KUKA KRL program: firepit2_2.src

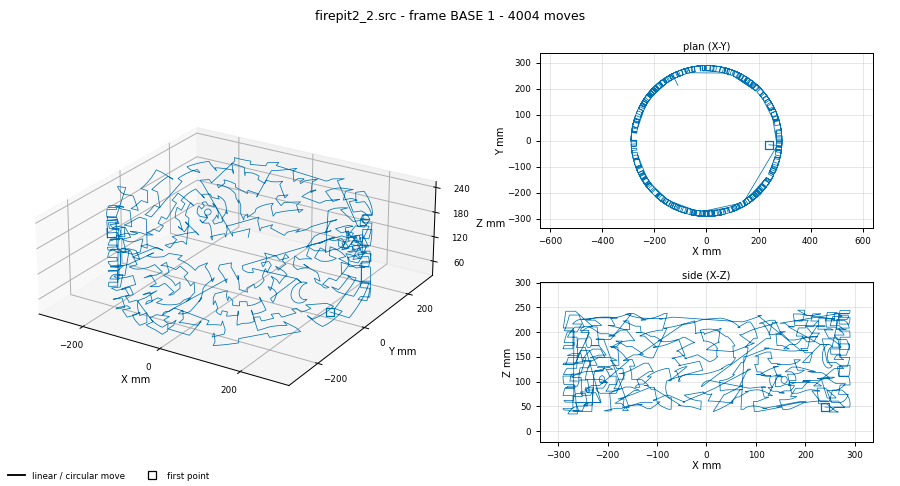
[picture p0: tool path of firepit2_2.src in frame BASE 1, 4004 of 4006 moves have a stored position in this frame; points joined in program order, loops and branches not executed]
&ACCESS RVP
&REL 1
&PARAM TEMPLATE = C:\KRC\Roboter\Template\vorgabe
&PARAM EDITMASK = *
DEF firepit2_2( )
EXT BAS (BAS_COMMAND :IN,REAL :IN )
DECL EKI_STATUS RET

INT INDX
FOR INDX=1 TO 6
	$ACC_AXIS[INDX]=50
	$VEL_AXIS[INDX]=20
ENDFOR

$VEL.ORI1=200
$VEL.ORI2=200
$ACC.ORI1=100
$ACC.ORI2=100

$VEL.CP = 0.1

$ACC.CP = 1

$IPO_MODE = #TCP
$APO.CDIS = 0.5
$ADVANCE = 5

$ACT_TOOL = 1
$TOOL=TOOL_DATA[1]
$ACT_BASE = 1
$BASE=BASE_DATA[1]

RET=EKI_Init("oxy")
RET=EKI_Open("oxy")

RET=EKI_SetBool("oxy","torchState",FALSE)
RET = EKI_Send("oxy","torchState")
PTP {A1 0.0,A2 -100.0,A3 150.0,A4 0.0,A5 -50.0,A6 0.0}

LIN {X 239.531,Y -14.995,Z 48.357,A 176.418,B 90.000,C 0.000} C_DIS
LIN {X 287.437,Y -17.994,Z 48.357,A 176.418,B 90.000,C 0.000} C_DIS
LIN {X 289.433,Y -18.119,Z 48.357,A 176.418,B 90.000,C 0.000} C_DIS
WAIT SEC 1.75
RET=EKI_SetBool("oxy","torchState",TRUE)
RET = EKI_Send("oxy","torchState")
LIN {X 289.566,Y -15.777,Z 49.221,A 176.881,B 90.000,C 0.000} C_DIS
LIN {X 289.684,Y -13.432,Z 50.078,A 177.345,B 90.000,C 0.000} C_DIS
LIN {X 289.787,Y -11.084,Z 50.930,A 177.810,B 90.000,C 0.000} C_DIS
LIN {X 289.865,Y -8.732,Z 51.772,A 178.274,B 90.000,C 0.000} C_DIS
LIN {X 289.925,Y -6.377,Z 52.608,A 178.740,B 90.000,C 0.000} C_DIS
LIN {X 289.970,Y -4.020,Z 53.438,A 179.206,B 90.000,C 0.000} C_DIS
LIN {X 289.992,Y -1.659,Z 54.260,A 179.672,B 90.000,C 0.000} C_DIS
LIN {X 289.994,Y 0.704,Z 55.074,A -179.861,B 90.000,C 0.000} C_DIS
LIN {X 289.981,Y 3.069,Z 55.883,A -179.394,B 90.000,C 0.000} C_DIS
LIN {X 289.946,Y 5.437,Z 56.685,A -178.926,B 90.000,C 0.000} C_DIS
LIN {X 289.890,Y 7.807,Z 57.478,A -178.457,B 90.000,C 0.000} C_DIS
LIN {X 289.818,Y 10.178,Z 58.266,A -177.989,B 90.000,C 0.000} C_DIS
LIN {X 289.726,Y 12.550,Z 59.048,A -177.520,B 90.000,C 0.000} C_DIS
LIN {X 289.610,Y 14.925,Z 59.821,A -177.050,B 90.000,C 0.000} C_DIS
LIN {X 289.480,Y 17.300,Z 60.589,A -176.580,B 90.000,C 0.000} C_DIS
LIN {X 289.329,Y 19.676,Z 61.350,A -176.110,B 90.000,C 0.000} C_DIS
LIN {X 289.155,Y 22.053,Z 62.103,A -175.639,B 90.000,C 0.000} C_DIS
LIN {X 288.966,Y 24.431,Z 62.851,A -175.167,B 90.000,C 0.000} C_DIS
LIN {X 288.755,Y 26.809,Z 63.592,A -174.696,B 90.000,C 0.000} C_DIS
LIN {X 288.522,Y 29.187,Z 64.326,A -174.224,B 90.000,C 0.000} C_DIS
LIN {X 288.274,Y 31.565,Z 65.055,A -173.751,B 90.000,C 0.000} C_DIS
LIN {X 288.003,Y 33.943,Z 65.776,A -173.278,B 90.000,C 0.000} C_DIS
LIN {X 287.711,Y 36.321,Z 66.491,A -172.805,B 90.000,C 0.000} C_DIS
LIN {X 287.405,Y 38.698,Z 67.201,A -172.331,B 90.000,C 0.000} C_DIS
LIN {X 287.072,Y 41.074,Z 67.903,A -171.857,B 90.000,C 0.000} C_DIS
LIN {X 286.721,Y 43.449,Z 68.599,A -171.383,B 90.000,C 0.000} C_DIS
LIN {X 286.357,Y 45.823,Z 69.290,A -170.909,B 90.000,C 0.000} C_DIS
LIN {X 285.961,Y 48.195,Z 69.973,A -170.433,B 90.000,C 0.000} C_DIS
LIN {X 285.553,Y 50.566,Z 70.651,A -169.958,B 90.000,C 0.000} C_DIS
LIN {X 285.125,Y 52.936,Z 71.323,A -169.482,B 90.000,C 0.000} C_DIS
LIN {X 284.672,Y 55.302,Z 71.988,A -169.006,B 90.000,C 0.000} C_DIS
LIN {X 284.205,Y 57.668,Z 72.649,A -168.530,B 90.000,C 0.000} C_DIS
LIN {X 283.714,Y 60.030,Z 73.302,A -168.053,B 90.000,C 0.000} C_DIS
LIN {X 283.203,Y 62.390,Z 73.949,A -167.576,B 90.000,C 0.000} C_DIS
LIN {X 282.679,Y 64.747,Z 74.593,A -167.099,B 90.000,C 0.000} C_DIS
LIN {X 282.124,Y 67.101,Z 75.228,A -166.621,B 90.000,C 0.000} C_DIS
LIN {X 281.556,Y 69.452,Z 75.859,A -166.143,B 90.000,C 0.000} C_DIS
LIN {X 280.967,Y 71.799,Z 76.483,A -165.665,B 90.000,C 0.000} C_DIS
LIN {X 280.355,Y 74.143,Z 77.102,A -165.187,B 90.000,C 0.000} C_DIS
LIN {X 279.731,Y 76.484,Z 77.716,A -164.708,B 90.000,C 0.000} C_DIS
LIN {X 279.077,Y 78.819,Z 78.323,A -164.229,B 90.000,C 0.000} C_DIS
LIN {X 278.409,Y 81.151,Z 78.925,A -163.750,B 90.000,C 0.000} C_DIS
LIN {X 277.721,Y 83.479,Z 79.522,A -163.270,B 90.000,C 0.000} C_DIS
LIN {X 277.009,Y 85.802,Z 80.112,A -162.790,B 90.000,C 0.000} C_DIS
LIN {X 276.286,Y 88.121,Z 80.700,A -162.310,B 90.000,C 0.000} C_DIS
LIN {X 275.532,Y 90.433,Z 81.278,A -161.829,B 90.000,C 0.000} C_DIS
LIN {X 274.766,Y 92.742,Z 81.854,A -161.349,B 90.000,C 0.000} C_DIS
LIN {X 273.977,Y 95.045,Z 82.423,A -160.868,B 90.000,C 0.000} C_DIS
LIN {X 273.481,Y 96.479,Z 82.777,A -160.568,B 90.000,C 0.000} C_DIS
LIN {X 271.595,Y 95.814,Z 82.777,A -160.568,B 90.000,C 0.000} C_DIS
WAIT SEC 0.1
RET=EKI_SetBool("oxy","torchState",FALSE)
RET = EKI_Send("oxy","torchState")
LIN {X 254.620,Y 89.825,Z 82.777,A -160.568,B 90.000,C 0.000} C_DIS
LIN {X 248.225,Y 106.227,Z 60.394,A -156.832,B 90.000,C 0.000} C_DIS
LIN {X 264.774,Y 113.309,Z 60.394,A -156.832,B 90.000,C 0.000} C_DIS
LIN {X 266.612,Y 114.096,Z 60.394,A -156.832,B 90.000,C 0.000} C_DIS
WAIT SEC 1.75
RET=EKI_SetBool("oxy","torchState",TRUE)
RET = EKI_Send("oxy","torchState")
LIN {X 267.486,Y 112.033,Z 59.286,A -157.274,B 90.000,C 0.000} C_DIS
LIN {X 268.355,Y 109.934,Z 58.243,A -157.723,B 90.000,C 0.000} C_DIS
LIN {X 269.219,Y 107.802,Z 57.263,A -158.178,B 90.000,C 0.000} C_DIS
LIN {X 270.073,Y 105.642,Z 56.341,A -158.637,B 90.000,C 0.000} C_DIS
LIN {X 270.918,Y 103.455,Z 55.472,A -159.100,B 90.000,C 0.000} C_DIS
LIN {X 271.751,Y 101.246,Z 54.652,A -159.566,B 90.000,C 0.000} C_DIS
LIN {X 272.572,Y 99.017,Z 53.873,A -160.035,B 90.000,C 0.000} C_DIS
LIN {X 273.377,Y 96.768,Z 53.136,A -160.507,B 90.000,C 0.000} C_DIS
LIN {X 274.169,Y 94.505,Z 52.429,A -160.981,B 90.000,C 0.000} C_DIS
LIN {X 274.943,Y 92.226,Z 51.754,A -161.457,B 90.000,C 0.000} C_DIS
LIN {X 275.701,Y 89.937,Z 51.097,A -161.933,B 90.000,C 0.000} C_DIS
LIN {X 276.440,Y 87.636,Z 50.456,A -162.410,B 90.000,C 0.000} C_DIS
LIN {X 277.158,Y 85.327,Z 49.822,A -162.888,B 90.000,C 0.000} C_DIS
LIN {X 277.862,Y 83.014,Z 49.190,A -163.366,B 90.000,C 0.000} C_DIS
LIN {X 278.545,Y 80.695,Z 48.551,A -163.844,B 90.000,C 0.000} C_DIS
LIN {X 279.208,Y 78.374,Z 47.901,A -164.320,B 90.000,C 0.000} C_DIS
LIN {X 279.278,Y 78.127,Z 47.832,A -164.371,B 90.000,C 0.000} C_DIS
LIN {X 277.352,Y 77.589,Z 47.832,A -164.371,B 90.000,C 0.000} C_DIS
WAIT SEC 0.1
RET=EKI_SetBool("oxy","torchState",FALSE)
RET = EKI_Send("oxy","torchState")
LIN {X 260.017,Y 72.739,Z 47.832,A -164.371,B 90.000,C 0.000} C_DIS
LIN {X 247.948,Y 106.874,Z 38.411,A -156.682,B 90.000,C 0.000} C_DIS
LIN {X 264.477,Y 113.999,Z 38.411,A -156.682,B 90.000,C 0.000} C_DIS
LIN {X 266.314,Y 114.790,Z 38.411,A -156.682,B 90.000,C 0.000} C_DIS
WAIT SEC 1.75
RET=EKI_SetBool("oxy","torchState",TRUE)
RET = EKI_Send("oxy","torchState")
LIN {X 265.321,Y 117.066,Z 38.699,A -156.192,B 90.000,C 0.000} C_DIS
LIN {X 264.313,Y 119.326,Z 39.052,A -155.703,B 90.000,C 0.000} C_DIS
LIN {X 263.289,Y 121.568,Z 39.469,A -155.216,B 90.000,C 0.000} C_DIS
LIN {X 262.251,Y 123.791,Z 39.949,A -154.731,B 90.000,C 0.000} C_DIS
LIN {X 261.200,Y 125.993,Z 40.492,A -154.249,B 90.000,C 0.000} C_DIS
LIN {X 260.138,Y 128.173,Z 41.098,A -153.770,B 90.000,C 0.000} C_DIS
LIN {X 259.064,Y 130.330,Z 41.766,A -153.294,B 90.000,C 0.000} C_DIS
LIN {X 257.981,Y 132.461,Z 42.496,A -152.822,B 90.000,C 0.000} C_DIS
LIN {X 256.889,Y 134.566,Z 43.287,A -152.353,B 90.000,C 0.000} C_DIS
LIN {X 255.790,Y 136.643,Z 44.139,A -151.889,B 90.000,C 0.000} C_DIS
LIN {X 254.685,Y 138.691,Z 45.052,A -151.429,B 90.000,C 0.000} C_DIS
LIN {X 253.575,Y 140.710,Z 46.020,A -150.974,B 90.000,C 0.000} C_DIS
LIN {X 252.458,Y 142.705,Z 47.031,A -150.522,B 90.000,C 0.000} C_DIS
LIN {X 251.332,Y 144.678,Z 48.073,A -150.073,B 90.000,C 0.000} C_DIS
LIN {X 250.196,Y 146.635,Z 49.136,A -149.626,B 90.000,C 0.000} C_DIS
LIN {X 249.044,Y 148.578,Z 50.207,A -149.180,B 90.000,C 0.000} C_DIS
LIN {X 247.880,Y 150.515,Z 51.276,A -148.734,B 90.000,C 0.000} C_DIS
LIN {X 246.698,Y 152.447,Z 52.333,A -148.286,B 90.000,C 0.000} C_DIS
LIN {X 245.493,Y 154.379,Z 53.364,A -147.836,B 90.000,C 0.000} C_DIS
LIN {X 244.264,Y 156.316,Z 54.358,A -147.383,B 90.000,C 0.000} C_DIS
LIN {X 243.565,Y 157.405,Z 54.898,A -147.127,B 90.000,C 0.000} C_DIS
LIN {X 241.885,Y 156.319,Z 54.898,A -147.127,B 90.000,C 0.000} C_DIS
WAIT SEC 0.1
RET=EKI_SetBool("oxy","torchState",FALSE)
RET = EKI_Send("oxy","torchState")
LIN {X 226.767,Y 146.549,Z 54.898,A -147.127,B 90.000,C 0.000} C_DIS
LIN {X 223.466,Y 151.535,Z 86.695,A -145.858,B 90.000,C 0.000} C_DIS
LIN {X 238.364,Y 161.638,Z 86.695,A -145.858,B 90.000,C 0.000} C_DIS
LIN {X 240.019,Y 162.760,Z 86.695,A -145.858,B 90.000,C 0.000} C_DIS
WAIT SEC 1.75
RET=EKI_SetBool("oxy","torchState",TRUE)
RET = EKI_Send("oxy","torchState")
LIN {X 241.298,Y 160.857,Z 85.700,A -146.311,B 90.000,C 0.000} C_DIS
LIN {X 242.543,Y 158.973,Z 84.627,A -146.757,B 90.000,C 0.000} C_DIS
LIN {X 243.760,Y 157.100,Z 83.505,A -147.199,B 90.000,C 0.000} C_DIS
LIN {X 244.957,Y 155.226,Z 82.363,A -147.638,B 90.000,C 0.000} C_DIS
LIN {X 246.144,Y 153.340,Z 81.231,A -148.078,B 90.000,C 0.000} C_DIS
LIN {X 247.324,Y 151.429,Z 80.134,A -148.522,B 90.000,C 0.000} C_DIS
LIN {X 248.501,Y 149.489,Z 79.085,A -148.970,B 90.000,C 0.000} C_DIS
LIN {X 249.671,Y 147.527,Z 78.070,A -149.422,B 90.000,C 0.000} C_DIS
LIN {X 250.832,Y 145.544,Z 77.087,A -149.876,B 90.000,C 0.000} C_DIS
LIN {X 251.983,Y 143.543,Z 76.126,A -150.332,B 90.000,C 0.000} C_DIS
LIN {X 253.118,Y 141.527,Z 75.180,A -150.789,B 90.000,C 0.000} C_DIS
LIN {X 254.242,Y 139.502,Z 74.240,A -151.247,B 90.000,C 0.000} C_DIS
LIN {X 255.347,Y 137.467,Z 73.298,A -151.704,B 90.000,C 0.000} C_DIS
LIN {X 256.435,Y 135.428,Z 72.346,A -152.161,B 90.000,C 0.000} C_DIS
LIN {X 257.503,Y 133.386,Z 71.376,A -152.616,B 90.000,C 0.000} C_DIS
LIN {X 258.549,Y 131.346,Z 70.381,A -153.069,B 90.000,C 0.000} C_DIS
LIN {X 259.573,Y 129.311,Z 69.352,A -153.519,B 90.000,C 0.000} C_DIS
LIN {X 260.573,Y 127.285,Z 68.282,A -153.965,B 90.000,C 0.000} C_DIS
LIN {X 261.546,Y 125.273,Z 67.163,A -154.407,B 90.000,C 0.000} C_DIS
LIN {X 261.950,Y 124.427,Z 66.674,A -154.592,B 90.000,C 0.000} C_DIS
LIN {X 260.144,Y 123.569,Z 66.674,A -154.592,B 90.000,C 0.000} C_DIS
WAIT SEC 0.1
RET=EKI_SetBool("oxy","torchState",FALSE)
RET = EKI_Send("oxy","torchState")
LIN {X 243.885,Y 115.846,Z 66.674,A -154.592,B 90.000,C 0.000} C_DIS
LIN {X 231.327,Y 139.240,Z 107.204,A -148.956,B 90.000,C 0.000} C_DIS
LIN {X 246.749,Y 148.523,Z 107.204,A -148.956,B 90.000,C 0.000} C_DIS
LIN {X 248.462,Y 149.554,Z 107.204,A -148.956,B 90.000,C 0.000} C_DIS
WAIT SEC 1.75
RET=EKI_SetBool("oxy","torchState",TRUE)
RET = EKI_Send("oxy","torchState")
LIN {X 247.296,Y 151.473,Z 108.302,A -148.512,B 90.000,C 0.000} C_DIS
LIN {X 246.109,Y 153.394,Z 109.374,A -148.066,B 90.000,C 0.000} C_DIS
LIN {X 244.899,Y 155.319,Z 110.414,A -147.617,B 90.000,C 0.000} C_DIS
LIN {X 243.666,Y 157.247,Z 111.418,A -147.164,B 90.000,C 0.000} C_DIS
LIN {X 242.407,Y 159.180,Z 112.382,A -146.709,B 90.000,C 0.000} C_DIS
LIN {X 241.124,Y 161.117,Z 113.304,A -146.250,B 90.000,C 0.000} C_DIS
LIN {X 239.816,Y 163.059,Z 114.179,A -145.787,B 90.000,C 0.000} C_DIS
LIN {X 238.481,Y 165.005,Z 115.002,A -145.321,B 90.000,C 0.000} C_DIS
LIN {X 237.119,Y 166.956,Z 115.770,A -144.851,B 90.000,C 0.000} C_DIS
LIN {X 235.731,Y 168.910,Z 116.479,A -144.377,B 90.000,C 0.000} C_DIS
LIN {X 234.316,Y 170.867,Z 117.124,A -143.900,B 90.000,C 0.000} C_DIS
LIN {X 232.875,Y 172.826,Z 117.703,A -143.419,B 90.000,C 0.000} C_DIS
LIN {X 231.408,Y 174.786,Z 118.209,A -142.936,B 90.000,C 0.000} C_DIS
LIN {X 231.093,Y 175.203,Z 118.307,A -142.832,B 90.000,C 0.000} C_DIS
LIN {X 229.499,Y 173.994,Z 118.307,A -142.832,B 90.000,C 0.000} C_DIS
WAIT SEC 0.1
RET=EKI_SetBool("oxy","torchState",FALSE)
RET = EKI_Send("oxy","torchState")
LIN {X 215.156,Y 163.120,Z 118.307,A -142.832,B 90.000,C 0.000} C_DIS
LIN {X 204.521,Y 176.270,Z 120.528,A -139.243,B 90.000,C 0.000} C_DIS
LIN {X 218.156,Y 188.021,Z 120.528,A -139.243,B 90.000,C 0.000} C_DIS
LIN {X 219.671,Y 189.327,Z 120.528,A -139.243,B 90.000,C 0.000} C_DIS
WAIT SEC 1.75
RET=EKI_SetBool("oxy","torchState",TRUE)
RET = EKI_Send("oxy","torchState")
LIN {X 218.042,Y 191.198,Z 120.833,A -138.753,B 90.000,C 0.000} C_DIS
LIN {X 216.401,Y 193.054,Z 121.166,A -138.264,B 90.000,C 0.000} C_DIS
LIN {X 214.747,Y 194.893,Z 121.527,A -137.775,B 90.000,C 0.000} C_DIS
LIN {X 213.079,Y 196.714,Z 121.913,A -137.287,B 90.000,C 0.000} C_DIS
LIN {X 211.398,Y 198.519,Z 122.321,A -136.800,B 90.000,C 0.000} C_DIS
LIN {X 209.704,Y 200.307,Z 122.748,A -136.313,B 90.000,C 0.000} C_DIS
LIN {X 207.997,Y 202.078,Z 123.191,A -135.827,B 90.000,C 0.000} C_DIS
LIN {X 206.277,Y 203.833,Z 123.649,A -135.341,B 90.000,C 0.000} C_DIS
LIN {X 204.543,Y 205.572,Z 124.118,A -134.856,B 90.000,C 0.000} C_DIS
LIN {X 202.797,Y 207.295,Z 124.596,A -134.372,B 90.000,C 0.000} C_DIS
LIN {X 201.037,Y 209.004,Z 125.080,A -133.887,B 90.000,C 0.000} C_DIS
LIN {X 199.264,Y 210.696,Z 125.568,A -133.403,B 90.000,C 0.000} C_DIS
LIN {X 197.475,Y 212.372,Z 126.057,A -132.918,B 90.000,C 0.000} C_DIS
LIN {X 195.671,Y 214.032,Z 126.544,A -132.434,B 90.000,C 0.000} C_DIS
LIN {X 193.857,Y 215.682,Z 127.029,A -131.949,B 90.000,C 0.000} C_DIS
LIN {X 192.025,Y 217.315,Z 127.506,A -131.465,B 90.000,C 0.000} C_DIS
LIN {X 190.179,Y 218.934,Z 127.975,A -130.980,B 90.000,C 0.000} C_DIS
LIN {X 188.316,Y 220.537,Z 128.432,A -130.494,B 90.000,C 0.000} C_DIS
LIN {X 186.438,Y 222.126,Z 128.874,A -130.008,B 90.000,C 0.000} C_DIS
LIN {X 185.186,Y 223.173,Z 129.159,A -129.686,B 90.000,C 0.000} C_DIS
LIN {X 183.909,Y 221.633,Z 129.159,A -129.686,B 90.000,C 0.000} C_DIS
WAIT SEC 0.1
RET=EKI_SetBool("oxy","torchState",FALSE)
RET = EKI_Send("oxy","torchState")
LIN {X 172.415,Y 207.781,Z 129.159,A -129.686,B 90.000,C 0.000} C_DIS
LIN {X 158.887,Y 218.300,Z 119.669,A -126.049,B 90.000,C 0.000} C_DIS
LIN {X 169.480,Y 232.853,Z 119.669,A -126.049,B 90.000,C 0.000} C_DIS
LIN {X 170.657,Y 234.470,Z 119.669,A -126.049,B 90.000,C 0.000} C_DIS
WAIT SEC 1.75
RET=EKI_SetBool("oxy","torchState",TRUE)
RET = EKI_Send("oxy","torchState")
LIN {X 172.562,Y 233.072,Z 118.855,A -126.516,B 90.000,C 0.000} C_DIS
LIN {X 174.340,Y 231.745,Z 117.704,A -126.954,B 90.000,C 0.000} C_DIS
LIN {X 175.958,Y 230.518,Z 116.246,A -127.355,B 90.000,C 0.000} C_DIS
LIN {X 177.385,Y 229.422,Z 114.510,A -127.711,B 90.000,C 0.000} C_DIS
LIN {X 178.586,Y 228.489,Z 112.527,A -128.011,B 90.000,C 0.000} C_DIS
LIN {X 179.537,Y 227.742,Z 110.339,A -128.250,B 90.000,C 0.000} C_DIS
LIN {X 180.227,Y 227.197,Z 107.999,A -128.424,B 90.000,C 0.000} C_DIS
LIN {X 180.642,Y 226.867,Z 105.556,A -128.528,B 90.000,C 0.000} C_DIS
LIN {X 180.776,Y 226.760,Z 103.063,A -128.562,B 90.000,C 0.000} C_DIS
LIN {X 180.747,Y 226.783,Z 102.004,A -128.555,B 90.000,C 0.000} C_DIS
LIN {X 179.501,Y 225.219,Z 102.004,A -128.555,B 90.000,C 0.000} C_DIS
WAIT SEC 0.1
RET=EKI_SetBool("oxy","torchState",FALSE)
RET = EKI_Send("oxy","torchState")
LIN {X 168.282,Y 211.143,Z 102.004,A -128.555,B 90.000,C 0.000} C_DIS
LIN {X 165.577,Y 213.270,Z 91.649,A -127.825,B 90.000,C 0.000} C_DIS
LIN {X 176.616,Y 227.488,Z 91.649,A -127.825,B 90.000,C 0.000} C_DIS
LIN {X 177.842,Y 229.068,Z 91.649,A -127.825,B 90.000,C 0.000} C_DIS
WAIT SEC 1.75
RET=EKI_SetBool("oxy","torchState",TRUE)
RET = EKI_Send("oxy","torchState")
LIN {X 176.720,Y 229.935,Z 89.590,A -127.545,B 90.000,C 0.000} C_DIS
LIN {X 175.472,Y 230.889,Z 87.645,A -127.234,B 90.000,C 0.000} C_DIS
LIN {X 174.102,Y 231.923,Z 85.829,A -126.895,B 90.000,C 0.000} C_DIS
LIN {X 172.619,Y 233.030,Z 84.148,A -126.530,B 90.000,C 0.000} C_DIS
LIN {X 171.026,Y 234.201,Z 82.618,A -126.139,B 90.000,C 0.000} C_DIS
LIN {X 169.333,Y 235.428,Z 81.248,A -125.726,B 90.000,C 0.000} C_DIS
LIN {X 169.108,Y 235.590,Z 81.083,A -125.671,B 90.000,C 0.000} C_DIS
LIN {X 167.942,Y 233.965,Z 81.083,A -125.671,B 90.000,C 0.000} C_DIS
WAIT SEC 0.1
RET=EKI_SetBool("oxy","torchState",FALSE)
RET = EKI_Send("oxy","torchState")
LIN {X 157.445,Y 219.342,Z 81.083,A -125.671,B 90.000,C 0.000} C_DIS
LIN {X 146.229,Y 226.974,Z 76.881,A -122.792,B 90.000,C 0.000} C_DIS
LIN {X 155.977,Y 242.106,Z 76.881,A -122.792,B 90.000,C 0.000} C_DIS
LIN {X 157.060,Y 243.787,Z 76.881,A -122.792,B 90.000,C 0.000} C_DIS
WAIT SEC 1.75
RET=EKI_SetBool("oxy","torchState",TRUE)
RET = EKI_Send("oxy","torchState")
LIN {X 154.953,Y 245.131,Z 76.914,A -122.298,B 90.000,C 0.000} C_DIS
LIN {X 152.843,Y 246.453,Z 77.140,A -121.806,B 90.000,C 0.000} C_DIS
LIN {X 150.743,Y 247.743,Z 77.552,A -121.319,B 90.000,C 0.000} C_DIS
LIN {X 148.659,Y 248.998,Z 78.129,A -120.838,B 90.000,C 0.000} C_DIS
LIN {X 146.601,Y 250.216,Z 78.858,A -120.366,B 90.000,C 0.000} C_DIS
LIN {X 144.574,Y 251.393,Z 79.726,A -119.903,B 90.000,C 0.000} C_DIS
LIN {X 143.164,Y 252.199,Z 80.414,A -119.582,B 90.000,C 0.000} C_DIS
LIN {X 142.176,Y 250.459,Z 80.414,A -119.582,B 90.000,C 0.000} C_DIS
WAIT SEC 0.1
RET=EKI_SetBool("oxy","torchState",FALSE)
RET = EKI_Send("oxy","torchState")
LIN {X 133.290,Y 234.806,Z 80.414,A -119.582,B 90.000,C 0.000} C_DIS
LIN {X 124.077,Y 239.802,Z 88.044,A -117.358,B 90.000,C 0.000} C_DIS
LIN {X 132.349,Y 255.788,Z 88.044,A -117.358,B 90.000,C 0.000} C_DIS
LIN {X 133.268,Y 257.565,Z 88.044,A -117.358,B 90.000,C 0.000} C_DIS
WAIT SEC 1.75
RET=EKI_SetBool("oxy","torchState",TRUE)
RET = EKI_Send("oxy","torchState")
LIN {X 131.815,Y 258.311,Z 89.936,A -117.035,B 90.000,C 0.000} C_DIS
LIN {X 130.533,Y 258.962,Z 91.981,A -116.751,B 90.000,C 0.000} C_DIS
LIN {X 129.447,Y 259.506,Z 94.165,A -116.511,B 90.000,C 0.000} C_DIS
LIN {X 128.589,Y 259.932,Z 96.473,A -116.322,B 90.000,C 0.000} C_DIS
LIN {X 127.987,Y 260.229,Z 98.881,A -116.189,B 90.000,C 0.000} C_DIS
LIN {X 127.675,Y 260.383,Z 101.357,A -116.120,B 90.000,C 0.000} C_DIS
LIN {X 127.663,Y 260.388,Z 103.856,A -116.118,B 90.000,C 0.000} C_DIS
LIN {X 127.951,Y 260.247,Z 106.335,A -116.181,B 90.000,C 0.000} C_DIS
LIN {X 128.526,Y 259.964,Z 108.752,A -116.308,B 90.000,C 0.000} C_DIS
LIN {X 129.381,Y 259.539,Z 111.062,A -116.496,B 90.000,C 0.000} C_DIS
LIN {X 129.988,Y 259.236,Z 112.313,A -116.630,B 90.000,C 0.000} C_DIS
LIN {X 129.091,Y 257.448,Z 112.313,A -116.630,B 90.000,C 0.000} C_DIS
WAIT SEC 0.1
RET=EKI_SetBool("oxy","torchState",FALSE)
RET = EKI_Send("oxy","torchState")
LIN {X 121.023,Y 241.357,Z 112.313,A -116.630,B 90.000,C 0.000} C_DIS
LIN {X 100.815,Y 250.472,Z 114.333,A -111.925,B 90.000,C 0.000} C_DIS
LIN {X 107.536,Y 267.170,Z 114.333,A -111.925,B 90.000,C 0.000} C_DIS
LIN {X 108.283,Y 269.026,Z 114.333,A -111.925,B 90.000,C 0.000} C_DIS
WAIT SEC 1.75
RET=EKI_SetBool("oxy","torchState",TRUE)
RET = EKI_Send("oxy","torchState")
LIN {X 110.306,Y 268.202,Z 115.549,A -112.356,B 90.000,C 0.000} C_DIS
LIN {X 112.335,Y 267.358,Z 116.741,A -112.790,B 90.000,C 0.000} C_DIS
LIN {X 114.368,Y 266.495,Z 117.910,A -113.227,B 90.000,C 0.000} C_DIS
LIN {X 116.409,Y 265.610,Z 119.051,A -113.666,B 90.000,C 0.000} C_DIS
LIN {X 118.456,Y 264.703,Z 120.162,A -114.109,B 90.000,C 0.000} C_DIS
LIN {X 120.511,Y 263.774,Z 121.241,A -114.554,B 90.000,C 0.000} C_DIS
LIN {X 122.573,Y 262.822,Z 122.285,A -115.003,B 90.000,C 0.000} C_DIS
LIN {X 124.643,Y 261.847,Z 123.291,A -115.455,B 90.000,C 0.000} C_DIS
LIN {X 126.721,Y 260.848,Z 124.257,A -115.911,B 90.000,C 0.000} C_DIS
LIN {X 128.806,Y 259.825,Z 125.181,A -116.370,B 90.000,C 0.000} C_DIS
LIN {X 130.900,Y 258.776,Z 126.056,A -116.832,B 90.000,C 0.000} C_DIS
LIN {X 133.000,Y 257.702,Z 126.882,A -117.298,B 90.000,C 0.000} C_DIS
LIN {X 135.108,Y 256.604,Z 127.657,A -117.768,B 90.000,C 0.000} C_DIS
LIN {X 137.221,Y 255.480,Z 128.377,A -118.241,B 90.000,C 0.000} C_DIS
LIN {X 139.340,Y 254.330,Z 129.038,A -118.717,B 90.000,C 0.000} C_DIS
LIN {X 141.464,Y 253.155,Z 129.638,A -119.197,B 90.000,C 0.000} C_DIS
LIN {X 143.590,Y 251.955,Z 130.173,A -119.679,B 90.000,C 0.000} C_DIS
LIN {X 145.130,Y 251.072,Z 130.520,A -120.030,B 90.000,C 0.000} C_DIS
LIN {X 144.129,Y 249.341,Z 130.520,A -120.030,B 90.000,C 0.000} C_DIS
WAIT SEC 0.1
RET=EKI_SetBool("oxy","torchState",FALSE)
RET = EKI_Send("oxy","torchState")
LIN {X 135.121,Y 233.757,Z 130.520,A -120.030,B 90.000,C 0.000} C_DIS
LIN {X 143.559,Y 228.672,Z 109.790,A -122.120,B 90.000,C 0.000} C_DIS
LIN {X 153.130,Y 243.917,Z 109.790,A -122.120,B 90.000,C 0.000} C_DIS
LIN {X 154.193,Y 245.610,Z 109.790,A -122.120,B 90.000,C 0.000} C_DIS
WAIT SEC 1.75
RET=EKI_SetBool("oxy","torchState",TRUE)
RET = EKI_Send("oxy","torchState")
LIN {X 152.528,Y 246.648,Z 108.437,A -121.733,B 90.000,C 0.000} C_DIS
LIN {X 151.315,Y 247.394,Z 106.535,A -121.451,B 90.000,C 0.000} C_DIS
LIN {X 150.702,Y 247.768,Z 104.269,A -121.309,B 90.000,C 0.000} C_DIS
LIN {X 150.768,Y 247.728,Z 101.911,A -121.325,B 90.000,C 0.000} C_DIS
LIN {X 151.506,Y 247.277,Z 99.699,A -121.496,B 90.000,C 0.000} C_DIS
LIN {X 152.817,Y 246.469,Z 97.891,A -121.800,B 90.000,C 0.000} C_DIS
LIN {X 154.590,Y 245.361,Z 96.642,A -122.213,B 90.000,C 0.000} C_DIS
LIN {X 156.542,Y 244.120,Z 96.120,A -122.670,B 90.000,C 0.000} C_DIS
LIN {X 158.530,Y 242.834,Z 96.324,A -123.138,B 90.000,C 0.000} C_DIS
LIN {X 160.361,Y 241.628,Z 97.241,A -123.571,B 90.000,C 0.000} C_DIS
LIN {X 161.850,Y 240.633,Z 98.788,A -123.925,B 90.000,C 0.000} C_DIS
LIN {X 162.847,Y 239.960,Z 100.839,A -124.162,B 90.000,C 0.000} C_DIS
LIN {X 163.218,Y 239.708,Z 103.053,A -124.251,B 90.000,C 0.000} C_DIS
LIN {X 162.986,Y 239.866,Z 105.293,A -124.196,B 90.000,C 0.000} C_DIS
LIN {X 162.127,Y 240.447,Z 107.414,A -123.991,B 90.000,C 0.000} C_DIS
LIN {X 160.737,Y 241.379,Z 109.093,A -123.660,B 90.000,C 0.000} C_DIS
LIN {X 158.968,Y 242.547,Z 110.164,A -123.241,B 90.000,C 0.000} C_DIS
LIN {X 156.974,Y 243.842,Z 110.535,A -122.771,B 90.000,C 0.000} C_DIS
LIN {X 154.998,Y 245.103,Z 110.166,A -122.308,B 90.000,C 0.000} C_DIS
LIN {X 154.193,Y 245.610,Z 109.790,A -122.120,B 90.000,C 0.000} C_DIS
LIN {X 153.130,Y 243.917,Z 109.790,A -122.120,B 90.000,C 0.000} C_DIS
WAIT SEC 0.1
RET=EKI_SetBool("oxy","torchState",FALSE)
RET = EKI_Send("oxy","torchState")
LIN {X 143.559,Y 228.672,Z 109.790,A -122.120,B 90.000,C 0.000} C_DIS
LIN {X 124.325,Y 239.673,Z 71.385,A -117.417,B 90.000,C 0.000} C_DIS
LIN {X 132.614,Y 255.651,Z 71.385,A -117.417,B 90.000,C 0.000} C_DIS
LIN {X 133.535,Y 257.427,Z 71.385,A -117.417,B 90.000,C 0.000} C_DIS
WAIT SEC 1.75
RET=EKI_SetBool("oxy","torchState",TRUE)
RET = EKI_Send("oxy","torchState")
LIN {X 131.536,Y 258.452,Z 72.482,A -116.973,B 90.000,C 0.000} C_DIS
LIN {X 129.535,Y 259.460,Z 73.591,A -116.531,B 90.000,C 0.000} C_DIS
LIN {X 127.528,Y 260.454,Z 74.701,A -116.088,B 90.000,C 0.000} C_DIS
LIN {X 125.509,Y 261.433,Z 75.801,A -115.645,B 90.000,C 0.000} C_DIS
LIN {X 123.472,Y 262.402,Z 76.878,A -115.199,B 90.000,C 0.000} C_DIS
LIN {X 121.411,Y 263.361,Z 77.918,A -114.750,B 90.000,C 0.000} C_DIS
LIN {X 119.324,Y 264.314,Z 78.911,A -114.297,B 90.000,C 0.000} C_DIS
LIN {X 117.204,Y 265.260,Z 79.839,A -113.838,B 90.000,C 0.000} C_DIS
LIN {X 115.050,Y 266.201,Z 80.689,A -113.374,B 90.000,C 0.000} C_DIS
LIN {X 112.860,Y 267.138,Z 81.448,A -112.903,B 90.000,C 0.000} C_DIS
LIN {X 110.632,Y 268.068,Z 82.095,A -112.426,B 90.000,C 0.000} C_DIS
LIN {X 108.369,Y 268.991,Z 82.617,A -111.943,B 90.000,C 0.000} C_DIS
LIN {X 106.073,Y 269.904,Z 82.999,A -111.455,B 90.000,C 0.000} C_DIS
LIN {X 104.619,Y 270.472,Z 83.162,A -111.147,B 90.000,C 0.000} C_DIS
LIN {X 103.898,Y 268.606,Z 83.162,A -111.147,B 90.000,C 0.000} C_DIS
WAIT SEC 0.1
RET=EKI_SetBool("oxy","torchState",FALSE)
RET = EKI_Send("oxy","torchState")
LIN {X 97.404,Y 251.818,Z 83.162,A -111.147,B 90.000,C 0.000} C_DIS
LIN {X 78.406,Y 258.365,Z 79.461,A -106.881,B 90.000,C 0.000} C_DIS
LIN {X 83.633,Y 275.590,Z 79.461,A -106.881,B 90.000,C 0.000} C_DIS
LIN {X 84.213,Y 277.503,Z 79.461,A -106.881,B 90.000,C 0.000} C_DIS
WAIT SEC 1.75
RET=EKI_SetBool("oxy","torchState",TRUE)
RET = EKI_Send("oxy","torchState")
LIN {X 82.009,Y 278.162,Z 78.484,A -106.427,B 90.000,C 0.000} C_DIS
LIN {X 79.833,Y 278.795,Z 77.428,A -105.979,B 90.000,C 0.000} C_DIS
LIN {X 77.686,Y 279.401,Z 76.299,A -105.538,B 90.000,C 0.000} C_DIS
LIN {X 75.569,Y 279.981,Z 75.104,A -105.105,B 90.000,C 0.000} C_DIS
LIN {X 73.479,Y 280.537,Z 73.851,A -104.677,B 90.000,C 0.000} C_DIS
LIN {X 71.413,Y 281.070,Z 72.549,A -104.256,B 90.000,C 0.000} C_DIS
LIN {X 69.370,Y 281.580,Z 71.202,A -103.840,B 90.000,C 0.000} C_DIS
LIN {X 67.345,Y 282.071,Z 69.821,A -103.428,B 90.000,C 0.000} C_DIS
LIN {X 65.653,Y 282.471,Z 68.637,A -103.085,B 90.000,C 0.000} C_DIS
LIN {X 65.200,Y 280.523,Z 68.637,A -103.085,B 90.000,C 0.000} C_DIS
WAIT SEC 0.1
RET=EKI_SetBool("oxy","torchState",FALSE)
RET = EKI_Send("oxy","torchState")
LIN {X 61.125,Y 262.990,Z 68.637,A -103.085,B 90.000,C 0.000} C_DIS
LIN {X 50.456,Y 265.244,Z 60.394,A -100.770,B 90.000,C 0.000} C_DIS
LIN {X 53.820,Y 282.927,Z 60.394,A -100.770,B 90.000,C 0.000} C_DIS
LIN {X 54.194,Y 284.891,Z 60.394,A -100.770,B 90.000,C 0.000} C_DIS
WAIT SEC 1.75
RET=EKI_SetBool("oxy","torchState",TRUE)
RET = EKI_Send("oxy","torchState")
LIN {X 52.155,Y 285.271,Z 58.998,A -100.361,B 90.000,C 0.000} C_DIS
LIN {X 50.097,Y 285.640,Z 57.628,A -99.948,B 90.000,C 0.000} C_DIS
LIN {X 48.018,Y 285.996,Z 56.286,A -99.531,B 90.000,C 0.000} C_DIS
LIN {X 45.920,Y 286.340,Z 54.971,A -99.111,B 90.000,C 0.000} C_DIS
LIN {X 43.804,Y 286.672,Z 53.683,A -98.688,B 90.000,C 0.000} C_DIS
LIN {X 41.668,Y 286.990,Z 52.424,A -98.261,B 90.000,C 0.000} C_DIS
LIN {X 39.515,Y 287.295,Z 51.191,A -97.831,B 90.000,C 0.000} C_DIS
LIN {X 37.342,Y 287.585,Z 49.990,A -97.398,B 90.000,C 0.000} C_DIS
LIN {X 35.153,Y 287.861,Z 48.814,A -96.962,B 90.000,C 0.000} C_DIS
LIN {X 32.947,Y 288.122,Z 47.669,A -96.523,B 90.000,C 0.000} C_DIS
LIN {X 30.724,Y 288.367,Z 46.552,A -96.082,B 90.000,C 0.000} C_DIS
LIN {X 28.486,Y 288.597,Z 45.462,A -95.637,B 90.000,C 0.000} C_DIS
LIN {X 26.231,Y 288.810,Z 44.405,A -95.190,B 90.000,C 0.000} C_DIS
LIN {X 23.963,Y 289.008,Z 43.374,A -94.740,B 90.000,C 0.000} C_DIS
LIN {X 21.678,Y 289.188,Z 42.375,A -94.287,B 90.000,C 0.000} C_DIS
LIN {X 19.380,Y 289.351,Z 41.405,A -93.832,B 90.000,C 0.000} C_DIS
LIN {X 17.069,Y 289.497,Z 40.464,A -93.374,B 90.000,C 0.000} C_DIS
LIN {X 14.835,Y 289.620,Z 39.588,A -92.932,B 90.000,C 0.000} C_DIS
LIN {X 14.733,Y 287.623,Z 39.588,A -92.932,B 90.000,C 0.000} C_DIS
WAIT SEC 0.1
RET=EKI_SetBool("oxy","torchState",FALSE)
RET = EKI_Send("oxy","torchState")
LIN {X 13.812,Y 269.646,Z 39.588,A -92.932,B 90.000,C 0.000} C_DIS
LIN {X 35.731,Y 267.625,Z 74.127,A -97.605,B 90.000,C 0.000} C_DIS
LIN {X 38.113,Y 285.467,Z 74.127,A -97.605,B 90.000,C 0.000} C_DIS
LIN {X 38.378,Y 287.449,Z 74.127,A -97.605,B 90.000,C 0.000} C_DIS
WAIT SEC 1.75
RET=EKI_SetBool("oxy","torchState",TRUE)
RET = EKI_Send("oxy","torchState")
LIN {X 40.577,Y 287.147,Z 75.275,A -98.043,B 90.000,C 0.000} C_DIS
LIN {X 42.781,Y 286.826,Z 76.411,A -98.483,B 90.000,C 0.000} C_DIS
LIN {X 44.987,Y 286.488,Z 77.536,A -98.924,B 90.000,C 0.000} C_DIS
LIN {X 47.195,Y 286.133,Z 78.653,A -99.366,B 90.000,C 0.000} C_DIS
LIN {X 49.403,Y 285.757,Z 79.763,A -99.809,B 90.000,C 0.000} C_DIS
LIN {X 51.609,Y 285.367,Z 80.873,A -100.251,B 90.000,C 0.000} C_DIS
LIN {X 53.812,Y 284.964,Z 81.982,A -100.694,B 90.000,C 0.000} C_DIS
LIN {X 56.010,Y 284.535,Z 83.093,A -101.136,B 90.000,C 0.000} C_DIS
LIN {X 58.204,Y 284.096,Z 84.207,A -101.578,B 90.000,C 0.000} C_DIS
LIN {X 60.392,Y 283.641,Z 85.327,A -102.020,B 90.000,C 0.000} C_DIS
LIN {X 62.572,Y 283.169,Z 86.456,A -102.460,B 90.000,C 0.000} C_DIS
LIN {X 64.742,Y 282.681,Z 87.596,A -102.900,B 90.000,C 0.000} C_DIS
LIN {X 66.901,Y 282.177,Z 88.752,A -103.338,B 90.000,C 0.000} C_DIS
LIN {X 69.047,Y 281.659,Z 89.923,A -103.774,B 90.000,C 0.000} C_DIS
LIN {X 71.180,Y 281.127,Z 91.114,A -104.208,B 90.000,C 0.000} C_DIS
LIN {X 72.146,Y 280.882,Z 91.659,A -104.405,B 90.000,C 0.000} C_DIS
LIN {X 71.649,Y 278.945,Z 91.659,A -104.405,B 90.000,C 0.000} C_DIS
WAIT SEC 0.1
RET=EKI_SetBool("oxy","torchState",FALSE)
RET = EKI_Send("oxy","torchState")
LIN {X 67.170,Y 261.511,Z 91.659,A -104.405,B 90.000,C 0.000} C_DIS
LIN {X 83.411,Y 256.793,Z 124.969,A -107.995,B 90.000,C 0.000} C_DIS
LIN {X 88.971,Y 273.913,Z 124.969,A -107.995,B 90.000,C 0.000} C_DIS
LIN {X 89.589,Y 275.815,Z 124.969,A -107.995,B 90.000,C 0.000} C_DIS
WAIT SEC 1.75
RET=EKI_SetBool("oxy","torchState",TRUE)
RET = EKI_Send("oxy","torchState")
LIN {X 87.456,Y 276.495,Z 123.858,A -107.552,B 90.000,C 0.000} C_DIS
LIN {X 85.318,Y 277.161,Z 122.747,A -107.110,B 90.000,C 0.000} C_DIS
LIN {X 83.176,Y 277.814,Z 121.635,A -106.667,B 90.000,C 0.000} C_DIS
LIN {X 81.031,Y 278.448,Z 120.519,A -106.226,B 90.000,C 0.000} C_DIS
LIN {X 78.881,Y 279.063,Z 119.403,A -105.784,B 90.000,C 0.000} C_DIS
LIN {X 76.728,Y 279.662,Z 118.283,A -105.342,B 90.000,C 0.000} C_DIS
LIN {X 74.572,Y 280.246,Z 117.161,A -104.901,B 90.000,C 0.000} C_DIS
LIN {X 72.411,Y 280.814,Z 116.039,A -104.459,B 90.000,C 0.000} C_DIS
LIN {X 70.249,Y 281.361,Z 114.912,A -104.019,B 90.000,C 0.000} C_DIS
LIN {X 68.082,Y 281.892,Z 113.784,A -103.578,B 90.000,C 0.000} C_DIS
LIN {X 65.913,Y 282.407,Z 112.653,A -103.138,B 90.000,C 0.000} C_DIS
LIN {X 63.742,Y 282.905,Z 111.519,A -102.697,B 90.000,C 0.000} C_DIS
LIN {X 61.567,Y 283.388,Z 110.384,A -102.257,B 90.000,C 0.000} C_DIS
LIN {X 59.392,Y 283.853,Z 109.244,A -101.818,B 90.000,C 0.000} C_DIS
LIN {X 57.213,Y 284.299,Z 108.104,A -101.378,B 90.000,C 0.000} C_DIS
LIN {X 55.031,Y 284.720,Z 106.959,A -100.939,B 90.000,C 0.000} C_DIS
LIN {X 52.849,Y 285.137,Z 105.812,A -100.500,B 90.000,C 0.000} C_DIS
LIN {X 50.665,Y 285.532,Z 104.662,A -100.062,B 90.000,C 0.000} C_DIS
LIN {X 48.480,Y 285.910,Z 103.509,A -99.624,B 90.000,C 0.000} C_DIS
LIN {X 46.293,Y 286.276,Z 102.354,A -99.186,B 90.000,C 0.000} C_DIS
LIN {X 44.105,Y 286.617,Z 101.195,A -98.748,B 90.000,C 0.000} C_DIS
LIN {X 41.917,Y 286.952,Z 100.034,A -98.311,B 90.000,C 0.000} C_DIS
LIN {X 39.727,Y 287.257,Z 98.868,A -97.874,B 90.000,C 0.000} C_DIS
LIN {X 37.537,Y 287.560,Z 97.701,A -97.437,B 90.000,C 0.000} C_DIS
LIN {X 35.346,Y 287.829,Z 96.528,A -97.001,B 90.000,C 0.000} C_DIS
LIN {X 33.155,Y 288.098,Z 95.355,A -96.565,B 90.000,C 0.000} C_DIS
LIN {X 30.964,Y 288.333,Z 94.175,A -96.130,B 90.000,C 0.000} C_DIS
LIN {X 28.773,Y 288.568,Z 92.995,A -95.694,B 90.000,C 0.000} C_DIS
LIN {X 26.582,Y 288.771,Z 91.808,A -95.259,B 90.000,C 0.000} C_DIS
LIN {X 24.392,Y 288.971,Z 90.621,A -94.825,B 90.000,C 0.000} C_DIS
LIN {X 22.202,Y 289.141,Z 89.427,A -94.391,B 90.000,C 0.000} C_DIS
LIN {X 20.013,Y 289.308,Z 88.233,A -93.957,B 90.000,C 0.000} C_DIS
LIN {X 17.825,Y 289.444,Z 87.031,A -93.524,B 90.000,C 0.000} C_DIS
LIN {X 15.637,Y 289.578,Z 85.830,A -93.091,B 90.000,C 0.000} C_DIS
LIN {X 14.130,Y 289.656,Z 84.998,A -92.793,B 90.000,C 0.000} C_DIS
LIN {X 14.032,Y 287.658,Z 84.998,A -92.793,B 90.000,C 0.000} C_DIS
WAIT SEC 0.1
RET=EKI_SetBool("oxy","torchState",FALSE)
RET = EKI_Send("oxy","torchState")
LIN {X 13.155,Y 269.679,Z 84.998,A -92.793,B 90.000,C 0.000} C_DIS
LIN {X -15.136,Y 269.575,Z 71.629,A -86.786,B 90.000,C 0.000} C_DIS
LIN {X -16.145,Y 287.547,Z 71.629,A -86.786,B 90.000,C 0.000} C_DIS
LIN {X -16.258,Y 289.544,Z 71.629,A -86.786,B 90.000,C 0.000} C_DIS
WAIT SEC 1.75
RET=EKI_SetBool("oxy","torchState",TRUE)
RET = EKI_Send("oxy","torchState")
LIN {X -18.555,Y 289.405,Z 70.655,A -86.331,B 90.000,C 0.000} C_DIS
LIN {X -20.852,Y 289.247,Z 69.681,A -85.877,B 90.000,C 0.000} C_DIS
LIN {X -23.148,Y 289.072,Z 68.707,A -85.422,B 90.000,C 0.000} C_DIS
LIN {X -25.442,Y 288.879,Z 67.733,A -84.967,B 90.000,C 0.000} C_DIS
LIN {X -27.734,Y 288.668,Z 66.759,A -84.512,B 90.000,C 0.000} C_DIS
LIN {X -30.025,Y 288.439,Z 65.785,A -84.057,B 90.000,C 0.000} C_DIS
LIN {X -32.314,Y 288.192,Z 64.811,A -83.602,B 90.000,C 0.000} C_DIS
LIN {X -34.600,Y 287.928,Z 63.837,A -83.148,B 90.000,C 0.000} C_DIS
LIN {X -36.885,Y 287.644,Z 62.863,A -82.693,B 90.000,C 0.000} C_DIS
LIN {X -39.167,Y 287.341,Z 61.889,A -82.238,B 90.000,C 0.000} C_DIS
LIN {X -41.447,Y 287.020,Z 60.915,A -81.783,B 90.000,C 0.000} C_DIS
LIN {X -43.724,Y 286.682,Z 59.941,A -81.328,B 90.000,C 0.000} C_DIS
LIN {X -45.998,Y 286.326,Z 58.967,A -80.873,B 90.000,C 0.000} C_DIS
LIN {X -47.443,Y 286.093,Z 58.348,A -80.584,B 90.000,C 0.000} C_DIS
LIN {X -47.116,Y 284.120,Z 58.348,A -80.584,B 90.000,C 0.000} C_DIS
WAIT SEC 0.1
RET=EKI_SetBool("oxy","torchState",FALSE)
RET = EKI_Send("oxy","torchState")
LIN {X -44.171,Y 266.362,Z 58.348,A -80.584,B 90.000,C 0.000} C_DIS
LIN {X -76.856,Y 258.830,Z 72.250,A -73.462,B 90.000,C 0.000} C_DIS
LIN {X -81.980,Y 276.086,Z 72.250,A -73.462,B 90.000,C 0.000} C_DIS
LIN {X -82.549,Y 278.003,Z 72.250,A -73.462,B 90.000,C 0.000} C_DIS
WAIT SEC 1.75
RET=EKI_SetBool("oxy","torchState",TRUE)
RET = EKI_Send("oxy","torchState")
LIN {X -84.747,Y 277.340,Z 71.262,A -73.008,B 90.000,C 0.000} C_DIS
LIN {X -86.939,Y 276.659,Z 70.270,A -72.555,B 90.000,C 0.000} C_DIS
LIN {X -89.127,Y 275.963,Z 69.283,A -72.101,B 90.000,C 0.000} C_DIS
LIN {X -91.314,Y 275.248,Z 68.307,A -71.647,B 90.000,C 0.000} C_DIS
LIN {X -93.504,Y 274.512,Z 67.350,A -71.190,B 90.000,C 0.000} C_DIS
LIN {X -95.698,Y 273.755,Z 66.422,A -70.732,B 90.000,C 0.000} C_DIS
LIN {X -97.899,Y 272.975,Z 65.531,A -70.270,B 90.000,C 0.000} C_DIS
LIN {X -100.109,Y 272.172,Z 64.683,A -69.806,B 90.000,C 0.000} C_DIS
LIN {X -102.330,Y 271.346,Z 63.887,A -69.338,B 90.000,C 0.000} C_DIS
LIN {X -104.563,Y 270.493,Z 63.154,A -68.865,B 90.000,C 0.000} C_DIS
LIN {X -106.807,Y 269.615,Z 62.491,A -68.389,B 90.000,C 0.000} C_DIS
LIN {X -107.768,Y 269.232,Z 62.230,A -68.185,B 90.000,C 0.000} C_DIS
LIN {X -107.025,Y 267.375,Z 62.230,A -68.185,B 90.000,C 0.000} C_DIS
WAIT SEC 0.1
RET=EKI_SetBool("oxy","torchState",FALSE)
RET = EKI_Send("oxy","torchState")
LIN {X -100.336,Y 250.664,Z 62.230,A -68.185,B 90.000,C 0.000} C_DIS
LIN {X -105.477,Y 248.545,Z 88.383,A -67.005,B 90.000,C 0.000} C_DIS
LIN {X -112.509,Y 265.115,Z 88.383,A -67.005,B 90.000,C 0.000} C_DIS
LIN {X -113.290,Y 266.956,Z 88.383,A -67.005,B 90.000,C 0.000} C_DIS
WAIT SEC 1.75
RET=EKI_SetBool("oxy","torchState",TRUE)
RET = EKI_Send("oxy","torchState")
LIN {X -115.441,Y 266.026,Z 87.512,A -66.542,B 90.000,C 0.000} C_DIS
LIN {X -117.588,Y 265.087,Z 86.643,A -66.079,B 90.000,C 0.000} C_DIS
LIN {X -119.728,Y 264.129,Z 85.776,A -65.615,B 90.000,C 0.000} C_DIS
LIN {X -121.861,Y 263.153,Z 84.913,A -65.152,B 90.000,C 0.000} C_DIS
LIN {X -123.987,Y 262.158,Z 84.053,A -64.688,B 90.000,C 0.000} C_DIS
LIN {X -126.107,Y 261.144,Z 83.199,A -64.224,B 90.000,C 0.000} C_DIS
LIN {X -128.219,Y 260.111,Z 82.350,A -63.760,B 90.000,C 0.000} C_DIS
LIN {X -130.325,Y 259.062,Z 81.507,A -63.295,B 90.000,C 0.000} C_DIS
LIN {X -132.424,Y 257.994,Z 80.671,A -62.829,B 90.000,C 0.000} C_DIS
LIN {X -134.519,Y 256.911,Z 79.840,A -62.363,B 90.000,C 0.000} C_DIS
LIN {X -136.606,Y 255.808,Z 79.017,A -61.897,B 90.000,C 0.000} C_DIS
LIN {X -138.685,Y 254.684,Z 78.205,A -61.430,B 90.000,C 0.000} C_DIS
LIN {X -140.760,Y 253.544,Z 77.400,A -60.962,B 90.000,C 0.000} C_DIS
LIN {X -142.827,Y 252.387,Z 76.604,A -60.494,B 90.000,C 0.000} C_DIS
LIN {X -144.889,Y 251.211,Z 75.819,A -60.025,B 90.000,C 0.000} C_DIS
LIN {X -146.943,Y 250.014,Z 75.046,A -59.556,B 90.000,C 0.000} C_DIS
LIN {X -148.990,Y 248.798,Z 74.285,A -59.085,B 90.000,C 0.000} C_DIS
LIN {X -151.031,Y 247.564,Z 73.536,A -58.614,B 90.000,C 0.000} C_DIS
LIN {X -153.065,Y 246.312,Z 72.800,A -58.142,B 90.000,C 0.000} C_DIS
LIN {X -155.092,Y 245.041,Z 72.077,A -57.669,B 90.000,C 0.000} C_DIS
LIN {X -157.113,Y 243.750,Z 71.369,A -57.196,B 90.000,C 0.000} C_DIS
LIN {X -159.126,Y 242.441,Z 70.676,A -56.721,B 90.000,C 0.000} C_DIS
LIN {X -161.132,Y 241.112,Z 69.998,A -56.246,B 90.000,C 0.000} C_DIS
LIN {X -163.131,Y 239.764,Z 69.337,A -55.769,B 90.000,C 0.000} C_DIS
LIN {X -165.122,Y 238.398,Z 68.693,A -55.292,B 90.000,C 0.000} C_DIS
LIN {X -167.106,Y 237.011,Z 68.067,A -54.814,B 90.000,C 0.000} C_DIS
LIN {X -169.082,Y 235.606,Z 67.459,A -54.335,B 90.000,C 0.000} C_DIS
LIN {X -171.050,Y 234.182,Z 66.870,A -53.855,B 90.000,C 0.000} C_DIS
LIN {X -173.010,Y 232.739,Z 66.301,A -53.374,B 90.000,C 0.000} C_DIS
LIN {X -174.961,Y 231.275,Z 65.754,A -52.892,B 90.000,C 0.000} C_DIS
LIN {X -176.903,Y 229.792,Z 65.228,A -52.409,B 90.000,C 0.000} C_DIS
LIN {X -178.838,Y 228.292,Z 64.722,A -51.926,B 90.000,C 0.000} C_DIS
LIN {X -178.859,Y 228.275,Z 64.716,A -51.920,B 90.000,C 0.000} C_DIS
LIN {X -177.626,Y 226.700,Z 64.716,A -51.920,B 90.000,C 0.000} C_DIS
WAIT SEC 0.1
RET=EKI_SetBool("oxy","torchState",FALSE)
RET = EKI_Send("oxy","torchState")
LIN {X -166.524,Y 212.532,Z 64.716,A -51.920,B 90.000,C 0.000} C_DIS
LIN {X -169.416,Y 210.234,Z 45.859,A -51.137,B 90.000,C 0.000} C_DIS
LIN {X -180.710,Y 224.249,Z 45.859,A -51.137,B 90.000,C 0.000} C_DIS
LIN {X -181.965,Y 225.807,Z 45.859,A -51.137,B 90.000,C 0.000} C_DIS
WAIT SEC 1.75
RET=EKI_SetBool("oxy","torchState",TRUE)
RET = EKI_Send("oxy","torchState")
LIN {X -183.893,Y 224.238,Z 45.586,A -50.646,B 90.000,C 0.000} C_DIS
LIN {X -185.805,Y 222.658,Z 45.283,A -50.155,B 90.000,C 0.000} C_DIS
LIN {X -187.699,Y 221.062,Z 44.947,A -49.666,B 90.000,C 0.000} C_DIS
LIN {X -189.578,Y 219.452,Z 44.586,A -49.177,B 90.000,C 0.000} C_DIS
LIN {X -191.440,Y 217.830,Z 44.203,A -48.689,B 90.000,C 0.000} C_DIS
LIN {X -193.287,Y 216.193,Z 43.801,A -48.202,B 90.000,C 0.000} C_DIS
LIN {X -195.117,Y 214.542,Z 43.384,A -47.715,B 90.000,C 0.000} C_DIS
LIN {X -196.931,Y 212.876,Z 42.957,A -47.228,B 90.000,C 0.000} C_DIS
LIN {X -198.730,Y 211.197,Z 42.523,A -46.742,B 90.000,C 0.000} C_DIS
LIN {X -200.516,Y 209.503,Z 42.086,A -46.256,B 90.000,C 0.000} C_DIS
LIN {X -202.289,Y 207.795,Z 41.652,A -45.769,B 90.000,C 0.000} C_DIS
LIN {X -204.047,Y 206.070,Z 41.228,A -45.283,B 90.000,C 0.000} C_DIS
LIN {X -205.793,Y 204.326,Z 40.826,A -44.795,B 90.000,C 0.000} C_DIS
LIN {X -206.893,Y 203.212,Z 40.585,A -44.486,B 90.000,C 0.000} C_DIS
LIN {X -205.467,Y 201.811,Z 40.585,A -44.486,B 90.000,C 0.000} C_DIS
WAIT SEC 0.1
RET=EKI_SetBool("oxy","torchState",FALSE)
RET = EKI_Send("oxy","torchState")
LIN {X -192.625,Y 189.197,Z 40.585,A -44.486,B 90.000,C 0.000} C_DIS
LIN {X -195.477,Y 186.249,Z 76.334,A -43.615,B 90.000,C 0.000} C_DIS
LIN {X -208.509,Y 198.665,Z 76.334,A -43.615,B 90.000,C 0.000} C_DIS
LIN {X -209.957,Y 200.045,Z 76.334,A -43.615,B 90.000,C 0.000} C_DIS
WAIT SEC 1.75
RET=EKI_SetBool("oxy","torchState",TRUE)
RET = EKI_Send("oxy","torchState")
LIN {X -211.660,Y 198.242,Z 76.027,A -43.125,B 90.000,C 0.000} C_DIS
LIN {X -213.361,Y 196.410,Z 76.035,A -42.631,B 90.000,C 0.000} C_DIS
LIN {X -215.031,Y 194.581,Z 76.377,A -42.142,B 90.000,C 0.000} C_DIS
LIN {X -216.636,Y 192.792,Z 77.063,A -41.667,B 90.000,C 0.000} C_DIS
LIN {X -218.143,Y 191.086,Z 78.096,A -41.217,B 90.000,C 0.000} C_DIS
LIN {X -219.528,Y 189.493,Z 79.435,A -40.800,B 90.000,C 0.000} C_DIS
LIN {X -220.788,Y 188.023,Z 81.017,A -40.418,B 90.000,C 0.000} C_DIS
LIN {X -221.927,Y 186.677,Z 82.788,A -40.069,B 90.000,C 0.000} C_DIS
LIN {X -222.958,Y 185.444,Z 84.703,A -39.752,B 90.000,C 0.000} C_DIS
LIN {X -223.864,Y 184.350,Z 86.663,A -39.471,B 90.000,C 0.000} C_DIS
LIN {X -222.320,Y 183.079,Z 86.663,A -39.471,B 90.000,C 0.000} C_DIS
WAIT SEC 0.1
RET=EKI_SetBool("oxy","torchState",FALSE)
RET = EKI_Send("oxy","torchState")
LIN {X -208.425,Y 171.636,Z 86.663,A -39.471,B 90.000,C 0.000} C_DIS
LIN {X -200.368,Y 180.977,Z 98.704,A -42.089,B 90.000,C 0.000} C_DIS
LIN {X -213.726,Y 193.042,Z 98.704,A -42.089,B 90.000,C 0.000} C_DIS
LIN {X -215.210,Y 194.382,Z 98.704,A -42.089,B 90.000,C 0.000} C_DIS
WAIT SEC 1.75
RET=EKI_SetBool("oxy","torchState",TRUE)
RET = EKI_Send("oxy","torchState")
LIN {X -213.892,Y 195.832,Z 97.152,A -42.476,B 90.000,C 0.000} C_DIS
LIN {X -212.304,Y 197.552,Z 96.275,A -42.939,B 90.000,C 0.000} C_DIS
LIN {X -210.596,Y 199.372,Z 96.142,A -43.432,B 90.000,C 0.000} C_DIS
LIN {X -208.924,Y 201.124,Z 96.762,A -43.910,B 90.000,C 0.000} C_DIS
LIN {X -207.449,Y 202.645,Z 98.088,A -44.329,B 90.000,C 0.000} C_DIS
LIN {X -206.327,Y 203.787,Z 100.008,A -44.645,B 90.000,C 0.000} C_DIS
LIN {X -205.710,Y 204.410,Z 102.217,A -44.818,B 90.000,C 0.000} C_DIS
LIN {X -205.603,Y 204.517,Z 104.588,A -44.848,B 90.000,C 0.000} C_DIS
LIN {X -206.018,Y 204.100,Z 106.878,A -44.732,B 90.000,C 0.000} C_DIS
LIN {X -206.908,Y 203.197,Z 108.886,A -44.481,B 90.000,C 0.000} C_DIS
LIN {X -208.248,Y 201.823,Z 110.488,A -44.102,B 90.000,C 0.000} C_DIS
LIN {X -209.854,Y 200.153,Z 111.425,A -43.644,B 90.000,C 0.000} C_DIS
LIN {X -211.567,Y 198.342,Z 111.621,A -43.152,B 90.000,C 0.000} C_DIS
LIN {X -213.225,Y 196.558,Z 111.062,A -42.671,B 90.000,C 0.000} C_DIS
LIN {X -214.678,Y 194.970,Z 109.791,A -42.246,B 90.000,C 0.000} C_DIS
LIN {X -215.737,Y 193.798,Z 108.026,A -41.934,B 90.000,C 0.000} C_DIS
LIN {X -216.387,Y 193.071,Z 105.859,A -41.741,B 90.000,C 0.000} C_DIS
LIN {X -216.559,Y 192.879,Z 103.511,A -41.690,B 90.000,C 0.000} C_DIS
LIN {X -216.237,Y 193.240,Z 101.193,A -41.786,B 90.000,C 0.000} C_DIS
LIN {X -215.452,Y 194.114,Z 99.129,A -42.018,B 90.000,C 0.000} C_DIS
LIN {X -215.210,Y 194.382,Z 98.704,A -42.089,B 90.000,C 0.000} C_DIS
LIN {X -213.726,Y 193.042,Z 98.704,A -42.089,B 90.000,C 0.000} C_DIS
WAIT SEC 0.1
RET=EKI_SetBool("oxy","torchState",FALSE)
RET = EKI_Send("oxy","torchState")
LIN {X -200.368,Y 180.977,Z 98.704,A -42.089,B 90.000,C 0.000} C_DIS
LIN {X -212.233,Y 166.905,Z 104.185,A -38.182,B 90.000,C 0.000} C_DIS
LIN {X -226.381,Y 178.032,Z 104.185,A -38.182,B 90.000,C 0.000} C_DIS
LIN {X -227.953,Y 179.269,Z 104.185,A -38.182,B 90.000,C 0.000} C_DIS
WAIT SEC 1.75
RET=EKI_SetBool("oxy","torchState",TRUE)
RET = EKI_Send("oxy","torchState")
LIN {X -228.024,Y 179.179,Z 106.682,A -38.160,B 90.000,C 0.000} C_DIS
LIN {X -227.968,Y 179.250,Z 109.180,A -38.178,B 90.000,C 0.000} C_DIS
LIN {X -227.782,Y 179.487,Z 111.662,A -38.237,B 90.000,C 0.000} C_DIS
LIN {X -227.463,Y 179.891,Z 114.108,A -38.339,B 90.000,C 0.000} C_DIS
LIN {X -227.010,Y 180.462,Z 116.499,A -38.483,B 90.000,C 0.000} C_DIS
LIN {X -226.418,Y 181.204,Z 118.811,A -38.671,B 90.000,C 0.000} C_DIS
LIN {X -225.685,Y 182.116,Z 121.020,A -38.902,B 90.000,C 0.000} C_DIS
LIN {X -225.217,Y 182.695,Z 122.193,A -39.049,B 90.000,C 0.000} C_DIS
LIN {X -223.663,Y 181.435,Z 122.193,A -39.049,B 90.000,C 0.000} C_DIS
WAIT SEC 0.1
RET=EKI_SetBool("oxy","torchState",FALSE)
RET = EKI_Send("oxy","torchState")
LIN {X -209.684,Y 170.095,Z 122.193,A -39.049,B 90.000,C 0.000} C_DIS
LIN {X -205.227,Y 175.447,Z 128.855,A -40.527,B 90.000,C 0.000} C_DIS
LIN {X -218.909,Y 187.144,Z 128.855,A -40.527,B 90.000,C 0.000} C_DIS
LIN {X -220.429,Y 188.443,Z 128.855,A -40.527,B 90.000,C 0.000} C_DIS
WAIT SEC 1.75
RET=EKI_SetBool("oxy","torchState",TRUE)
RET = EKI_Send("oxy","torchState")
LIN {X -218.898,Y 190.220,Z 129.720,A -40.990,B 90.000,C 0.000} C_DIS
LIN {X -217.281,Y 192.065,Z 130.193,A -41.475,B 90.000,C 0.000} C_DIS
LIN {X -215.618,Y 193.930,Z 130.266,A -41.969,B 90.000,C 0.000} C_DIS
LIN {X -214.060,Y 195.649,Z 129.965,A -42.427,B 90.000,C 0.000} C_DIS
LIN {X -212.583,Y 194.300,Z 129.965,A -42.427,B 90.000,C 0.000} C_DIS
WAIT SEC 0.1
RET=EKI_SetBool("oxy","torchState",FALSE)
RET = EKI_Send("oxy","torchState")
LIN {X -199.297,Y 182.156,Z 129.965,A -42.427,B 90.000,C 0.000} C_DIS
LIN {X -189.077,Y 192.743,Z 124.482,A -45.550,B 90.000,C 0.000} C_DIS
LIN {X -201.682,Y 205.592,Z 124.482,A -45.550,B 90.000,C 0.000} C_DIS
LIN {X -203.083,Y 207.020,Z 124.482,A -45.550,B 90.000,C 0.000} C_DIS
WAIT SEC 1.75
RET=EKI_SetBool("oxy","torchState",TRUE)
RET = EKI_Send("oxy","torchState")
LIN {X -201.704,Y 208.363,Z 122.886,A -45.930,B 90.000,C 0.000} C_DIS
LIN {X -200.429,Y 209.590,Z 121.121,A -46.280,B 90.000,C 0.000} C_DIS
LIN {X -199.268,Y 210.695,Z 119.202,A -46.597,B 90.000,C 0.000} C_DIS
LIN {X -198.231,Y 211.671,Z 117.148,A -46.878,B 90.000,C 0.000} C_DIS
LIN {X -197.330,Y 212.511,Z 114.973,A -47.121,B 90.000,C 0.000} C_DIS
LIN {X -196.575,Y 213.210,Z 112.695,A -47.325,B 90.000,C 0.000} C_DIS
LIN {X -196.082,Y 213.663,Z 110.815,A -47.457,B 90.000,C 0.000} C_DIS
LIN {X -194.729,Y 212.190,Z 110.815,A -47.457,B 90.000,C 0.000} C_DIS
WAIT SEC 0.1
RET=EKI_SetBool("oxy","torchState",FALSE)
RET = EKI_Send("oxy","torchState")
LIN {X -182.559,Y 198.928,Z 110.815,A -47.457,B 90.000,C 0.000} C_DIS
LIN {X -182.640,Y 198.853,Z 94.085,A -47.434,B 90.000,C 0.000} C_DIS
LIN {X -194.816,Y 212.110,Z 94.085,A -47.434,B 90.000,C 0.000} C_DIS
LIN {X -196.169,Y 213.583,Z 94.085,A -47.434,B 90.000,C 0.000} C_DIS
WAIT SEC 1.75
RET=EKI_SetBool("oxy","torchState",TRUE)
RET = EKI_Send("oxy","torchState")
LIN {X -196.826,Y 212.978,Z 91.750,A -47.257,B 90.000,C 0.000} C_DIS
LIN {X -197.635,Y 212.227,Z 89.507,A -47.039,B 90.000,C 0.000} C_DIS
LIN {X -198.586,Y 211.337,Z 87.374,A -46.782,B 90.000,C 0.000} C_DIS
LIN {X -199.668,Y 210.316,Z 85.365,A -46.488,B 90.000,C 0.000} C_DIS
LIN {X -200.872,Y 209.166,Z 83.500,A -46.159,B 90.000,C 0.000} C_DIS
LIN {X -202.185,Y 207.897,Z 81.794,A -45.798,B 90.000,C 0.000} C_DIS
LIN {X -203.305,Y 206.802,Z 80.556,A -45.489,B 90.000,C 0.000} C_DIS
LIN {X -201.903,Y 205.376,Z 80.556,A -45.489,B 90.000,C 0.000} C_DIS
WAIT SEC 0.1
RET=EKI_SetBool("oxy","torchState",FALSE)
RET = EKI_Send("oxy","torchState")
LIN {X -189.284,Y 192.540,Z 80.556,A -45.489,B 90.000,C 0.000} C_DIS
LIN {X -174.213,Y 206.276,Z 85.553,A -49.817,B 90.000,C 0.000} C_DIS
LIN {X -185.827,Y 220.028,Z 85.553,A -49.817,B 90.000,C 0.000} C_DIS
LIN {X -187.117,Y 221.556,Z 85.553,A -49.817,B 90.000,C 0.000} C_DIS
WAIT SEC 1.75
RET=EKI_SetBool("oxy","torchState",TRUE)
RET = EKI_Send("oxy","torchState")
LIN {X -185.762,Y 222.694,Z 87.318,A -50.167,B 90.000,C 0.000} C_DIS
LIN {X -184.502,Y 223.739,Z 89.208,A -50.490,B 90.000,C 0.000} C_DIS
LIN {X -183.346,Y 224.687,Z 91.211,A -50.785,B 90.000,C 0.000} C_DIS
LIN {X -182.301,Y 225.535,Z 93.317,A -51.051,B 90.000,C 0.000} C_DIS
LIN {X -181.371,Y 226.284,Z 95.514,A -51.287,B 90.000,C 0.000} C_DIS
LIN {X -180.564,Y 226.929,Z 97.790,A -51.491,B 90.000,C 0.000} C_DIS
LIN {X -179.885,Y 227.467,Z 100.135,A -51.662,B 90.000,C 0.000} C_DIS
LIN {X -179.339,Y 227.898,Z 102.536,A -51.800,B 90.000,C 0.000} C_DIS
LIN {X -178.992,Y 228.171,Z 104.572,A -51.887,B 90.000,C 0.000} C_DIS
LIN {X -177.757,Y 226.597,Z 104.572,A -51.887,B 90.000,C 0.000} C_DIS
WAIT SEC 0.1
RET=EKI_SetBool("oxy","torchState",FALSE)
RET = EKI_Send("oxy","torchState")
LIN {X -166.647,Y 212.435,Z 104.572,A -51.887,B 90.000,C 0.000} C_DIS
LIN {X -168.834,Y 210.701,Z 126.079,A -51.295,B 90.000,C 0.000} C_DIS
LIN {X -180.090,Y 224.748,Z 126.079,A -51.295,B 90.000,C 0.000} C_DIS
LIN {X -181.340,Y 226.309,Z 126.079,A -51.295,B 90.000,C 0.000} C_DIS
WAIT SEC 1.75
RET=EKI_SetBool("oxy","torchState",TRUE)
RET = EKI_Send("oxy","torchState")
LIN {X -182.269,Y 225.561,Z 128.276,A -51.059,B 90.000,C 0.000} C_DIS
LIN {X -183.314,Y 224.713,Z 130.383,A -50.794,B 90.000,C 0.000} C_DIS
LIN {X -184.466,Y 223.769,Z 132.390,A -50.499,B 90.000,C 0.000} C_DIS
LIN {X -185.716,Y 222.732,Z 134.290,A -50.178,B 90.000,C 0.000} C_DIS
LIN {X -187.054,Y 221.610,Z 136.079,A -49.833,B 90.000,C 0.000} C_DIS
LIN {X -188.470,Y 220.407,Z 137.752,A -49.466,B 90.000,C 0.000} C_DIS
LIN {X -189.955,Y 219.128,Z 139.303,A -49.079,B 90.000,C 0.000} C_DIS
LIN {X -191.501,Y 217.778,Z 140.729,A -48.673,B 90.000,C 0.000} C_DIS
LIN {X -193.102,Y 216.360,Z 142.025,A -48.251,B 90.000,C 0.000} C_DIS
LIN {X -194.039,Y 215.520,Z 142.707,A -48.002,B 90.000,C 0.000} C_DIS
LIN {X -192.701,Y 214.033,Z 142.707,A -48.002,B 90.000,C 0.000} C_DIS
WAIT SEC 0.1
RET=EKI_SetBool("oxy","torchState",FALSE)
RET = EKI_Send("oxy","torchState")
LIN {X -180.657,Y 200.656,Z 142.707,A -48.002,B 90.000,C 0.000} C_DIS
LIN {X -192.799,Y 189.020,Z 148.285,A -44.433,B 90.000,C 0.000} C_DIS
LIN {X -205.652,Y 201.621,Z 148.285,A -44.433,B 90.000,C 0.000} C_DIS
LIN {X -207.081,Y 203.021,Z 148.285,A -44.433,B 90.000,C 0.000} C_DIS
WAIT SEC 1.75
RET=EKI_SetBool("oxy","torchState",TRUE)
RET = EKI_Send("oxy","torchState")
LIN {X -208.802,Y 201.251,Z 148.674,A -43.945,B 90.000,C 0.000} C_DIS
LIN {X -210.514,Y 199.458,Z 148.995,A -43.455,B 90.000,C 0.000} C_DIS
LIN {X -212.218,Y 197.645,Z 149.236,A -42.964,B 90.000,C 0.000} C_DIS
LIN {X -213.910,Y 195.812,Z 149.387,A -42.471,B 90.000,C 0.000} C_DIS
LIN {X -215.590,Y 193.961,Z 149.433,A -41.977,B 90.000,C 0.000} C_DIS
LIN {X -217.253,Y 192.096,Z 149.363,A -41.483,B 90.000,C 0.000} C_DIS
LIN {X -218.896,Y 190.223,Z 149.162,A -40.991,B 90.000,C 0.000} C_DIS
LIN {X -220.429,Y 188.443,Z 148.840,A -40.527,B 90.000,C 0.000} C_DIS
LIN {X -218.909,Y 187.144,Z 148.840,A -40.527,B 90.000,C 0.000} C_DIS
WAIT SEC 0.1
RET=EKI_SetBool("oxy","torchState",FALSE)
RET = EKI_Send("oxy","torchState")
LIN {X -205.227,Y 175.447,Z 148.840,A -40.527,B 90.000,C 0.000} C_DIS
LIN {X -214.002,Y 164.631,Z 165.495,A -37.571,B 90.000,C 0.000} C_DIS
LIN {X -228.269,Y 175.606,Z 165.495,A -37.571,B 90.000,C 0.000} C_DIS
LIN {X -229.854,Y 176.825,Z 165.495,A -37.571,B 90.000,C 0.000} C_DIS
WAIT SEC 1.75
RET=EKI_SetBool("oxy","torchState",TRUE)
RET = EKI_Send("oxy","torchState")
LIN {X -231.279,Y 174.957,Z 164.643,A -37.107,B 90.000,C 0.000} C_DIS
LIN {X -232.679,Y 173.090,Z 163.748,A -36.646,B 90.000,C 0.000} C_DIS
LIN {X -234.054,Y 171.226,Z 162.806,A -36.188,B 90.000,C 0.000} C_DIS
LIN {X -235.402,Y 169.369,Z 161.816,A -35.735,B 90.000,C 0.000} C_DIS
LIN {X -236.722,Y 167.519,Z 160.774,A -35.286,B 90.000,C 0.000} C_DIS
LIN {X -238.013,Y 165.680,Z 159.679,A -34.842,B 90.000,C 0.000} C_DIS
LIN {X -239.274,Y 163.853,Z 158.530,A -34.403,B 90.000,C 0.000} C_DIS
LIN {X -240.505,Y 162.041,Z 157.325,A -33.970,B 90.000,C 0.000} C_DIS
LIN {X -241.703,Y 160.248,Z 156.061,A -33.544,B 90.000,C 0.000} C_DIS
LIN {X -242.869,Y 158.477,Z 154.738,A -33.125,B 90.000,C 0.000} C_DIS
LIN {X -243.999,Y 156.731,Z 153.351,A -32.714,B 90.000,C 0.000} C_DIS
LIN {X -245.093,Y 155.014,Z 151.901,A -32.312,B 90.000,C 0.000} C_DIS
LIN {X -246.150,Y 153.329,Z 150.387,A -31.919,B 90.000,C 0.000} C_DIS
LIN {X -247.170,Y 151.681,Z 148.808,A -31.536,B 90.000,C 0.000} C_DIS
LIN {X -248.148,Y 150.075,Z 147.160,A -31.165,B 90.000,C 0.000} C_DIS
LIN {X -249.085,Y 148.515,Z 145.447,A -30.805,B 90.000,C 0.000} C_DIS
LIN {X -249.979,Y 147.005,Z 143.667,A -30.458,B 90.000,C 0.000} C_DIS
LIN {X -250.419,Y 146.255,Z 142.734,A -30.287,B 90.000,C 0.000} C_DIS
LIN {X -248.692,Y 145.246,Z 142.734,A -30.287,B 90.000,C 0.000} C_DIS
WAIT SEC 0.1
RET=EKI_SetBool("oxy","torchState",FALSE)
RET = EKI_Send("oxy","torchState")
LIN {X -233.149,Y 136.168,Z 142.734,A -30.287,B 90.000,C 0.000} C_DIS
LIN {X -237.772,Y 127.924,Z 127.745,A -28.281,B 90.000,C 0.000} C_DIS
LIN {X -253.623,Y 136.453,Z 127.745,A -28.281,B 90.000,C 0.000} C_DIS
LIN {X -255.384,Y 137.400,Z 127.745,A -28.281,B 90.000,C 0.000} C_DIS
WAIT SEC 1.75
RET=EKI_SetBool("oxy","torchState",TRUE)
RET = EKI_Send("oxy","torchState")
LIN {X -255.873,Y 136.487,Z 125.470,A -28.076,B 90.000,C 0.000} C_DIS
LIN {X -256.315,Y 135.656,Z 123.154,A -27.890,B 90.000,C 0.000} C_DIS
LIN {X -256.706,Y 134.914,Z 120.799,A -27.725,B 90.000,C 0.000} C_DIS
LIN {X -257.048,Y 134.263,Z 118.410,A -27.579,B 90.000,C 0.000} C_DIS
LIN {X -257.339,Y 133.704,Z 115.991,A -27.455,B 90.000,C 0.000} C_DIS
LIN {X -257.576,Y 133.247,Z 113.545,A -27.353,B 90.000,C 0.000} C_DIS
LIN {X -257.760,Y 132.890,Z 111.077,A -27.274,B 90.000,C 0.000} C_DIS
LIN {X -257.890,Y 132.638,Z 108.594,A -27.218,B 90.000,C 0.000} C_DIS
LIN {X -257.963,Y 132.496,Z 106.099,A -27.186,B 90.000,C 0.000} C_DIS
LIN {X -257.977,Y 132.468,Z 103.600,A -27.180,B 90.000,C 0.000} C_DIS
LIN {X -257.972,Y 132.477,Z 102.963,A -27.182,B 90.000,C 0.000} C_DIS
LIN {X -256.193,Y 131.564,Z 102.963,A -27.182,B 90.000,C 0.000} C_DIS
WAIT SEC 0.1
RET=EKI_SetBool("oxy","torchState",FALSE)
RET = EKI_Send("oxy","torchState")
LIN {X -240.181,Y 123.341,Z 102.963,A -27.182,B 90.000,C 0.000} C_DIS
LIN {X -236.822,Y 129.673,Z 78.891,A -28.703,B 90.000,C 0.000} C_DIS
LIN {X -252.611,Y 138.318,Z 78.891,A -28.703,B 90.000,C 0.000} C_DIS
LIN {X -254.365,Y 139.279,Z 78.891,A -28.703,B 90.000,C 0.000} C_DIS
WAIT SEC 1.75
RET=EKI_SetBool("oxy","torchState",TRUE)
RET = EKI_Send("oxy","torchState")
LIN {X -253.641,Y 140.592,Z 76.891,A -28.999,B 90.000,C 0.000} C_DIS
LIN {X -252.851,Y 142.008,Z 74.988,A -29.320,B 90.000,C 0.000} C_DIS
LIN {X -251.996,Y 143.519,Z 73.190,A -29.663,B 90.000,C 0.000} C_DIS
LIN {X -251.490,Y 144.405,Z 72.229,A -29.864,B 90.000,C 0.000} C_DIS
LIN {X -249.756,Y 143.409,Z 72.229,A -29.864,B 90.000,C 0.000} C_DIS
WAIT SEC 0.1
RET=EKI_SetBool("oxy","torchState",FALSE)
RET = EKI_Send("oxy","torchState")
LIN {X -234.146,Y 134.446,Z 72.229,A -29.864,B 90.000,C 0.000} C_DIS
LIN {X -227.974,Y 144.665,Z 87.218,A -32.398,B 90.000,C 0.000} C_DIS
LIN {X -243.172,Y 154.310,Z 87.218,A -32.398,B 90.000,C 0.000} C_DIS
LIN {X -244.860,Y 155.381,Z 87.218,A -32.398,B 90.000,C 0.000} C_DIS
WAIT SEC 1.75
RET=EKI_SetBool("oxy","torchState",TRUE)
RET = EKI_Send("oxy","torchState")
LIN {X -244.340,Y 156.199,Z 84.914,A -32.589,B 90.000,C 0.000} C_DIS
LIN {X -243.658,Y 157.260,Z 82.756,A -32.839,B 90.000,C 0.000} C_DIS
LIN {X -242.824,Y 158.545,Z 80.780,A -33.141,B 90.000,C 0.000} C_DIS
LIN {X -241.851,Y 160.026,Z 79.018,A -33.492,B 90.000,C 0.000} C_DIS
LIN {X -240.747,Y 161.682,Z 77.505,A -33.885,B 90.000,C 0.000} C_DIS
LIN {X -240.665,Y 161.803,Z 77.408,A -33.914,B 90.000,C 0.000} C_DIS
LIN {X -239.005,Y 160.687,Z 77.408,A -33.914,B 90.000,C 0.000} C_DIS
WAIT SEC 0.1
RET=EKI_SetBool("oxy","torchState",FALSE)
RET = EKI_Send("oxy","torchState")
LIN {X -224.068,Y 150.644,Z 77.408,A -33.914,B 90.000,C 0.000} C_DIS
LIN {X -214.306,Y 164.234,Z 57.820,A -37.465,B 90.000,C 0.000} C_DIS
LIN {X -228.593,Y 175.183,Z 57.820,A -37.465,B 90.000,C 0.000} C_DIS
LIN {X -230.181,Y 176.400,Z 57.820,A -37.465,B 90.000,C 0.000} C_DIS
WAIT SEC 1.75
RET=EKI_SetBool("oxy","torchState",TRUE)
RET = EKI_Send("oxy","torchState")
LIN {X -231.688,Y 174.406,Z 57.771,A -36.971,B 90.000,C 0.000} C_DIS
LIN {X -233.182,Y 172.402,Z 57.727,A -36.477,B 90.000,C 0.000} C_DIS
LIN {X -234.662,Y 170.388,Z 57.688,A -35.983,B 90.000,C 0.000} C_DIS
LIN {X -236.117,Y 168.356,Z 57.656,A -35.490,B 90.000,C 0.000} C_DIS
LIN {X -237.565,Y 166.319,Z 57.626,A -34.996,B 90.000,C 0.000} C_DIS
LIN {X -238.983,Y 164.260,Z 57.604,A -34.502,B 90.000,C 0.000} C_DIS
LIN {X -240.397,Y 162.199,Z 57.582,A -34.008,B 90.000,C 0.000} C_DIS
LIN {X -241.787,Y 160.121,Z 57.566,A -33.514,B 90.000,C 0.000} C_DIS
LIN {X -243.157,Y 158.031,Z 57.549,A -33.020,B 90.000,C 0.000} C_DIS
LIN {X -244.507,Y 155.927,Z 57.537,A -32.526,B 90.000,C 0.000} C_DIS
LIN {X -245.843,Y 153.814,Z 57.525,A -32.033,B 90.000,C 0.000} C_DIS
LIN {X -247.163,Y 151.691,Z 57.514,A -31.539,B 90.000,C 0.000} C_DIS
LIN {X -248.459,Y 149.554,Z 57.503,A -31.045,B 90.000,C 0.000} C_DIS
LIN {X -249.738,Y 147.406,Z 57.493,A -30.551,B 90.000,C 0.000} C_DIS
LIN {X -250.996,Y 145.246,Z 57.481,A -30.057,B 90.000,C 0.000} C_DIS
LIN {X -252.239,Y 143.077,Z 57.468,A -29.563,B 90.000,C 0.000} C_DIS
LIN {X -253.465,Y 140.899,Z 57.454,A -29.069,B 90.000,C 0.000} C_DIS
LIN {X -254.673,Y 138.711,Z 57.438,A -28.575,B 90.000,C 0.000} C_DIS
LIN {X -255.860,Y 136.511,Z 57.418,A -28.082,B 90.000,C 0.000} C_DIS
LIN {X -257.027,Y 134.300,Z 57.395,A -27.588,B 90.000,C 0.000} C_DIS
LIN {X -258.175,Y 132.080,Z 57.368,A -27.094,B 90.000,C 0.000} C_DIS
LIN {X -259.304,Y 129.850,Z 57.336,A -26.600,B 90.000,C 0.000} C_DIS
LIN {X -260.407,Y 127.607,Z 57.297,A -26.106,B 90.000,C 0.000} C_DIS
LIN {X -261.504,Y 125.361,Z 57.257,A -25.612,B 90.000,C 0.000} C_DIS
LIN {X -261.901,Y 124.530,Z 57.240,A -25.430,B 90.000,C 0.000} C_DIS
LIN {X -260.095,Y 123.672,Z 57.240,A -25.430,B 90.000,C 0.000} C_DIS
WAIT SEC 0.1
RET=EKI_SetBool("oxy","torchState",FALSE)
RET = EKI_Send("oxy","torchState")
LIN {X -243.839,Y 115.942,Z 57.240,A -25.430,B 90.000,C 0.000} C_DIS
LIN {X -251.171,Y 99.062,Z 40.585,A -21.524,B 90.000,C 0.000} C_DIS
LIN {X -267.915,Y 105.666,Z 40.585,A -21.524,B 90.000,C 0.000} C_DIS
LIN {X -269.776,Y 106.400,Z 40.585,A -21.524,B 90.000,C 0.000} C_DIS
WAIT SEC 1.75
RET=EKI_SetBool("oxy","torchState",TRUE)
RET = EKI_Send("oxy","torchState")
LIN {X -268.848,Y 108.721,Z 40.631,A -22.018,B 90.000,C 0.000} C_DIS
LIN {X -267.901,Y 111.034,Z 40.661,A -22.512,B 90.000,C 0.000} C_DIS
LIN {X -266.934,Y 113.339,Z 40.676,A -23.006,B 90.000,C 0.000} C_DIS
LIN {X -265.948,Y 115.636,Z 40.675,A -23.500,B 90.000,C 0.000} C_DIS
LIN {X -264.940,Y 117.924,Z 40.659,A -23.994,B 90.000,C 0.000} C_DIS
LIN {X -263.913,Y 120.202,Z 40.630,A -24.487,B 90.000,C 0.000} C_DIS
LIN {X -262.866,Y 122.472,Z 40.589,A -24.981,B 90.000,C 0.000} C_DIS
LIN {X -261.800,Y 124.732,Z 40.537,A -25.475,B 90.000,C 0.000} C_DIS
LIN {X -260.717,Y 126.984,Z 40.475,A -25.969,B 90.000,C 0.000} C_DIS
LIN {X -259.615,Y 129.227,Z 40.403,A -26.462,B 90.000,C 0.000} C_DIS
LIN {X -258.488,Y 131.457,Z 40.320,A -26.956,B 90.000,C 0.000} C_DIS
LIN {X -257.349,Y 133.680,Z 40.233,A -27.450,B 90.000,C 0.000} C_DIS
LIN {X -256.189,Y 135.892,Z 40.137,A -27.943,B 90.000,C 0.000} C_DIS
LIN {X -255.010,Y 138.094,Z 40.035,A -28.437,B 90.000,C 0.000} C_DIS
LIN {X -253.804,Y 140.281,Z 39.927,A -28.930,B 90.000,C 0.000} C_DIS
LIN {X -252.591,Y 142.464,Z 39.817,A -29.423,B 90.000,C 0.000} C_DIS
LIN {X -251.357,Y 144.635,Z 39.702,A -29.917,B 90.000,C 0.000} C_DIS
LIN {X -250.095,Y 146.789,Z 39.584,A -30.410,B 90.000,C 0.000} C_DIS
LIN {X -248.924,Y 148.785,Z 39.475,A -30.867,B 90.000,C 0.000} C_DIS
LIN {X -247.207,Y 147.759,Z 39.475,A -30.867,B 90.000,C 0.000} C_DIS
WAIT SEC 0.1
RET=EKI_SetBool("oxy","torchState",FALSE)
RET = EKI_Send("oxy","torchState")
LIN {X -231.757,Y 138.524,Z 39.475,A -30.867,B 90.000,C 0.000} C_DIS
LIN {X -227.974,Y 144.665,Z 103.873,A -32.398,B 90.000,C 0.000} C_DIS
LIN {X -243.172,Y 154.310,Z 103.873,A -32.398,B 90.000,C 0.000} C_DIS
LIN {X -244.860,Y 155.381,Z 103.873,A -32.398,B 90.000,C 0.000} C_DIS
WAIT SEC 1.75
RET=EKI_SetBool("oxy","torchState",TRUE)
RET = EKI_Send("oxy","torchState")
LIN {X -244.552,Y 155.866,Z 106.306,A -32.512,B 90.000,C 0.000} C_DIS
LIN {X -244.202,Y 156.414,Z 108.719,A -32.640,B 90.000,C 0.000} C_DIS
LIN {X -243.808,Y 157.027,Z 111.111,A -32.784,B 90.000,C 0.000} C_DIS
LIN {X -243.369,Y 157.708,Z 113.475,A -32.944,B 90.000,C 0.000} C_DIS
LIN {X -242.883,Y 158.454,Z 115.811,A -33.120,B 90.000,C 0.000} C_DIS
LIN {X -242.350,Y 159.269,Z 118.113,A -33.312,B 90.000,C 0.000} C_DIS
LIN {X -241.766,Y 160.153,Z 120.377,A -33.522,B 90.000,C 0.000} C_DIS
LIN {X -241.133,Y 161.106,Z 122.600,A -33.748,B 90.000,C 0.000} C_DIS
LIN {X -240.445,Y 162.130,Z 124.774,A -33.991,B 90.000,C 0.000} C_DIS
LIN {X -239.705,Y 163.222,Z 126.897,A -34.252,B 90.000,C 0.000} C_DIS
LIN {X -238.909,Y 164.385,Z 128.961,A -34.531,B 90.000,C 0.000} C_DIS
LIN {X -238.056,Y 165.618,Z 130.962,A -34.827,B 90.000,C 0.000} C_DIS
LIN {X -237.197,Y 166.846,Z 132.791,A -35.123,B 90.000,C 0.000} C_DIS
LIN {X -235.561,Y 165.695,Z 132.791,A -35.123,B 90.000,C 0.000} C_DIS
WAIT SEC 0.1
RET=EKI_SetBool("oxy","torchState",FALSE)
RET = EKI_Send("oxy","torchState")
LIN {X -220.839,Y 155.339,Z 132.791,A -35.123,B 90.000,C 0.000} C_DIS
LIN {X -236.682,Y 129.929,Z 162.850,A -28.765,B 90.000,C 0.000} C_DIS
LIN {X -252.461,Y 138.591,Z 162.850,A -28.765,B 90.000,C 0.000} C_DIS
LIN {X -254.214,Y 139.553,Z 162.850,A -28.765,B 90.000,C 0.000} C_DIS
WAIT SEC 1.75
RET=EKI_SetBool("oxy","torchState",TRUE)
RET = EKI_Send("oxy","torchState")
LIN {X -255.103,Y 137.923,Z 161.177,A -28.398,B 90.000,C 0.000} C_DIS
LIN {X -255.966,Y 136.311,Z 159.472,A -28.037,B 90.000,C 0.000} C_DIS
LIN {X -256.814,Y 134.706,Z 157.754,A -27.678,B 90.000,C 0.000} C_DIS
LIN {X -257.653,Y 133.096,Z 156.035,A -27.320,B 90.000,C 0.000} C_DIS
LIN {X -258.487,Y 131.470,Z 154.330,A -26.958,B 90.000,C 0.000} C_DIS
LIN {X -259.324,Y 129.810,Z 152.659,A -26.591,B 90.000,C 0.000} C_DIS
LIN {X -260.169,Y 128.108,Z 151.035,A -26.216,B 90.000,C 0.000} C_DIS
LIN {X -261.027,Y 126.352,Z 149.476,A -25.830,B 90.000,C 0.000} C_DIS
LIN {X -261.466,Y 125.441,Z 148.718,A -25.630,B 90.000,C 0.000} C_DIS
LIN {X -259.663,Y 124.576,Z 148.718,A -25.630,B 90.000,C 0.000} C_DIS
WAIT SEC 0.1
RET=EKI_SetBool("oxy","torchState",FALSE)
RET = EKI_Send("oxy","torchState")
LIN {X -243.434,Y 116.790,Z 148.718,A -25.630,B 90.000,C 0.000} C_DIS
LIN {X -254.153,Y 91.139,Z 115.023,A -19.728,B 90.000,C 0.000} C_DIS
LIN {X -271.096,Y 97.215,Z 115.023,A -19.728,B 90.000,C 0.000} C_DIS
LIN {X -272.979,Y 97.890,Z 115.023,A -19.728,B 90.000,C 0.000} C_DIS
WAIT SEC 1.75
RET=EKI_SetBool("oxy","torchState",TRUE)
RET = EKI_Send("oxy","torchState")
LIN {X -273.421,Y 96.648,Z 112.899,A -19.467,B 90.000,C 0.000} C_DIS
LIN {X -273.867,Y 95.376,Z 110.794,A -19.201,B 90.000,C 0.000} C_DIS
LIN {X -274.321,Y 94.065,Z 108.715,A -18.927,B 90.000,C 0.000} C_DIS
LIN {X -274.783,Y 92.704,Z 106.669,A -18.643,B 90.000,C 0.000} C_DIS
LIN {X -275.257,Y 91.287,Z 104.665,A -18.348,B 90.000,C 0.000} C_DIS
LIN {X -275.745,Y 89.802,Z 102.715,A -18.039,B 90.000,C 0.000} C_DIS
LIN {X -276.210,Y 88.363,Z 100.964,A -17.740,B 90.000,C 0.000} C_DIS
LIN {X -274.305,Y 87.754,Z 100.964,A -17.740,B 90.000,C 0.000} C_DIS
WAIT SEC 0.1
RET=EKI_SetBool("oxy","torchState",FALSE)
RET = EKI_Send("oxy","torchState")
LIN {X -257.161,Y 82.269,Z 100.964,A -17.740,B 90.000,C 0.000} C_DIS
LIN {X -260.764,Y 70.016,Z 90.620,A -15.030,B 90.000,C 0.000} C_DIS
LIN {X -278.148,Y 74.684,Z 90.620,A -15.030,B 90.000,C 0.000} C_DIS
LIN {X -280.080,Y 75.203,Z 90.620,A -15.030,B 90.000,C 0.000} C_DIS
WAIT SEC 1.75
RET=EKI_SetBool("oxy","torchState",TRUE)
RET = EKI_Send("oxy","torchState")
LIN {X -280.674,Y 72.952,Z 89.708,A -14.570,B 90.000,C 0.000} C_DIS
LIN {X -281.265,Y 70.638,Z 88.972,A -14.098,B 90.000,C 0.000} C_DIS
LIN {X -281.849,Y 68.273,Z 88.411,A -13.617,B 90.000,C 0.000} C_DIS
LIN {X -282.420,Y 65.871,Z 88.017,A -13.129,B 90.000,C 0.000} C_DIS
LIN {X -282.974,Y 63.446,Z 87.781,A -12.637,B 90.000,C 0.000} C_DIS
LIN {X -283.510,Y 61.005,Z 87.695,A -12.144,B 90.000,C 0.000} C_DIS
LIN {X -284.026,Y 58.560,Z 87.753,A -11.650,B 90.000,C 0.000} C_DIS
LIN {X -284.518,Y 56.117,Z 87.945,A -11.158,B 90.000,C 0.000} C_DIS
LIN {X -284.725,Y 55.061,Z 88.068,A -10.945,B 90.000,C 0.000} C_DIS
LIN {X -282.761,Y 54.681,Z 88.068,A -10.945,B 90.000,C 0.000} C_DIS
WAIT SEC 0.1
RET=EKI_SetBool("oxy","torchState",FALSE)
RET = EKI_Send("oxy","torchState")
LIN {X -265.089,Y 51.263,Z 88.068,A -10.945,B 90.000,C 0.000} C_DIS
LIN {X -268.005,Y 32.758,Z 94.110,A -6.969,B 90.000,C 0.000} C_DIS
LIN {X -285.872,Y 34.942,Z 94.110,A -6.969,B 90.000,C 0.000} C_DIS
LIN {X -287.858,Y 35.184,Z 94.110,A -6.969,B 90.000,C 0.000} C_DIS
WAIT SEC 1.75
RET=EKI_SetBool("oxy","torchState",TRUE)
RET = EKI_Send("oxy","torchState")
LIN {X -288.124,Y 32.923,Z 95.142,A -6.519,B 90.000,C 0.000} C_DIS
LIN {X -288.372,Y 30.676,Z 96.208,A -6.072,B 90.000,C 0.000} C_DIS
LIN {X -288.601,Y 28.440,Z 97.302,A -5.628,B 90.000,C 0.000} C_DIS
LIN {X -288.812,Y 26.212,Z 98.416,A -5.186,B 90.000,C 0.000} C_DIS
LIN {X -289.004,Y 23.989,Z 99.542,A -4.745,B 90.000,C 0.000} C_DIS
LIN {X -289.179,Y 21.765,Z 100.671,A -4.304,B 90.000,C 0.000} C_DIS
LIN {X -289.340,Y 19.540,Z 101.798,A -3.864,B 90.000,C 0.000} C_DIS
LIN {X -289.483,Y 17.308,Z 102.915,A -3.422,B 90.000,C 0.000} C_DIS
LIN {X -289.608,Y 15.066,Z 104.013,A -2.978,B 90.000,C 0.000} C_DIS
LIN {X -289.717,Y 12.810,Z 105.083,A -2.532,B 90.000,C 0.000} C_DIS
LIN {X -289.808,Y 10.536,Z 106.117,A -2.082,B 90.000,C 0.000} C_DIS
LIN {X -289.882,Y 8.243,Z 107.110,A -1.629,B 90.000,C 0.000} C_DIS
LIN {X -289.939,Y 5.928,Z 108.051,A -1.171,B 90.000,C 0.000} C_DIS
LIN {X -289.977,Y 3.588,Z 108.929,A -0.709,B 90.000,C 0.000} C_DIS
LIN {X -289.997,Y 1.222,Z 109.738,A -0.241,B 90.000,C 0.000} C_DIS
LIN {X -289.997,Y -1.169,Z 110.467,A 0.231,B 90.000,C 0.000} C_DIS
LIN {X -289.982,Y -3.272,Z 111.033,A 0.647,B 90.000,C 0.000} C_DIS
LIN {X -287.982,Y -3.250,Z 111.033,A 0.647,B 90.000,C 0.000} C_DIS
WAIT SEC 0.1
RET=EKI_SetBool("oxy","torchState",FALSE)
RET = EKI_Send("oxy","torchState")
LIN {X -269.983,Y -3.047,Z 111.033,A 0.647,B 90.000,C 0.000} C_DIS
LIN {X -269.212,Y -20.615,Z 114.173,A 4.379,B 90.000,C 0.000} C_DIS
LIN {X -287.159,Y -21.990,Z 114.173,A 4.379,B 90.000,C 0.000} C_DIS
LIN {X -289.153,Y -22.142,Z 114.173,A 4.379,B 90.000,C 0.000} C_DIS
WAIT SEC 1.75
RET=EKI_SetBool("oxy","torchState",TRUE)
RET = EKI_Send("oxy","torchState")
LIN {X -288.954,Y -24.600,Z 114.584,A 4.866,B 90.000,C 0.000} C_DIS
LIN {X -288.735,Y -27.050,Z 115.031,A 5.352,B 90.000,C 0.000} C_DIS
LIN {X -288.496,Y -29.490,Z 115.516,A 5.837,B 90.000,C 0.000} C_DIS
LIN {X -288.237,Y -31.922,Z 116.032,A 6.320,B 90.000,C 0.000} C_DIS
LIN {X -287.958,Y -34.345,Z 116.582,A 6.802,B 90.000,C 0.000} C_DIS
LIN {X -287.660,Y -36.759,Z 117.158,A 7.282,B 90.000,C 0.000} C_DIS
LIN {X -287.342,Y -39.164,Z 117.762,A 7.761,B 90.000,C 0.000} C_DIS
LIN {X -287.005,Y -41.559,Z 118.391,A 8.239,B 90.000,C 0.000} C_DIS
LIN {X -286.649,Y -43.947,Z 119.040,A 8.716,B 90.000,C 0.000} C_DIS
LIN {X -286.274,Y -46.326,Z 119.709,A 9.192,B 90.000,C 0.000} C_DIS
LIN {X -285.880,Y -48.697,Z 120.394,A 9.667,B 90.000,C 0.000} C_DIS
LIN {X -285.467,Y -51.061,Z 121.094,A 10.141,B 90.000,C 0.000} C_DIS
LIN {X -285.035,Y -53.418,Z 121.807,A 10.615,B 90.000,C 0.000} C_DIS
LIN {X -284.583,Y -55.768,Z 122.529,A 11.087,B 90.000,C 0.000} C_DIS
LIN {X -284.115,Y -58.113,Z 123.258,A 11.560,B 90.000,C 0.000} C_DIS
LIN {X -283.625,Y -60.451,Z 123.994,A 12.032,B 90.000,C 0.000} C_DIS
LIN {X -283.118,Y -62.785,Z 124.732,A 12.504,B 90.000,C 0.000} C_DIS
LIN {X -282.592,Y -65.114,Z 125.471,A 12.976,B 90.000,C 0.000} C_DIS
LIN {X -282.049,Y -67.440,Z 126.209,A 13.447,B 90.000,C 0.000} C_DIS
LIN {X -281.647,Y -69.100,Z 126.735,A 13.785,B 90.000,C 0.000} C_DIS
LIN {X -279.705,Y -68.623,Z 126.735,A 13.785,B 90.000,C 0.000} C_DIS
WAIT SEC 0.1
RET=EKI_SetBool("oxy","torchState",FALSE)
RET = EKI_Send("oxy","torchState")
LIN {X -262.223,Y -64.334,Z 126.735,A 13.785,B 90.000,C 0.000} C_DIS
LIN {X -261.261,Y -68.137,Z 152.233,A 14.617,B 90.000,C 0.000} C_DIS
LIN {X -278.679,Y -72.679,Z 152.233,A 14.617,B 90.000,C 0.000} C_DIS
LIN {X -280.614,Y -73.184,Z 152.233,A 14.617,B 90.000,C 0.000} C_DIS
WAIT SEC 1.75
RET=EKI_SetBool("oxy","torchState",TRUE)
RET = EKI_Send("oxy","torchState")
LIN {X -279.985,Y -75.553,Z 152.723,A 15.101,B 90.000,C 0.000} C_DIS
LIN {X -279.333,Y -77.929,Z 153.145,A 15.588,B 90.000,C 0.000} C_DIS
LIN {X -278.658,Y -80.308,Z 153.514,A 16.077,B 90.000,C 0.000} C_DIS
LIN {X -277.961,Y -82.686,Z 153.839,A 16.566,B 90.000,C 0.000} C_DIS
LIN {X -277.244,Y -85.062,Z 154.139,A 17.057,B 90.000,C 0.000} C_DIS
LIN {X -276.504,Y -87.432,Z 154.425,A 17.547,B 90.000,C 0.000} C_DIS
LIN {X -275.746,Y -89.797,Z 154.712,A 18.038,B 90.000,C 0.000} C_DIS
LIN {X -274.969,Y -92.153,Z 155.014,A 18.528,B 90.000,C 0.000} C_DIS
LIN {X -274.171,Y -94.499,Z 155.345,A 19.018,B 90.000,C 0.000} C_DIS
LIN {X -273.355,Y -96.832,Z 155.721,A 19.506,B 90.000,C 0.000} C_DIS
LIN {X -272.524,Y -99.149,Z 156.152,A 19.992,B 90.000,C 0.000} C_DIS
LIN {X -272.343,Y -99.647,Z 156.251,A 20.097,B 90.000,C 0.000} C_DIS
LIN {X -270.464,Y -98.960,Z 156.251,A 20.097,B 90.000,C 0.000} C_DIS
WAIT SEC 0.1
RET=EKI_SetBool("oxy","torchState",FALSE)
RET = EKI_Send("oxy","torchState")
LIN {X -253.560,Y -92.775,Z 156.251,A 20.097,B 90.000,C 0.000} C_DIS
LIN {X -249.816,Y -102.430,Z 136.942,A 22.295,B 90.000,C 0.000} C_DIS
LIN {X -266.471,Y -109.259,Z 136.942,A 22.295,B 90.000,C 0.000} C_DIS
LIN {X -268.321,Y -110.017,Z 136.942,A 22.295,B 90.000,C 0.000} C_DIS
WAIT SEC 1.75
RET=EKI_SetBool("oxy","torchState",TRUE)
RET = EKI_Send("oxy","torchState")
LIN {X -267.368,Y -112.311,Z 137.223,A 22.785,B 90.000,C 0.000} C_DIS
LIN {X -266.395,Y -114.600,Z 137.469,A 23.277,B 90.000,C 0.000} C_DIS
LIN {X -265.400,Y -116.884,Z 137.683,A 23.769,B 90.000,C 0.000} C_DIS
LIN {X -264.386,Y -119.160,Z 137.875,A 24.261,B 90.000,C 0.000} C_DIS
LIN {X -263.351,Y -121.429,Z 138.048,A 24.754,B 90.000,C 0.000} C_DIS
LIN {X -262.295,Y -123.689,Z 138.211,A 25.247,B 90.000,C 0.000} C_DIS
LIN {X -261.222,Y -125.941,Z 138.371,A 25.740,B 90.000,C 0.000} C_DIS
LIN {X -260.131,Y -128.184,Z 138.531,A 26.233,B 90.000,C 0.000} C_DIS
LIN {X -259.019,Y -130.417,Z 138.700,A 26.725,B 90.000,C 0.000} C_DIS
LIN {X -257.889,Y -132.639,Z 138.884,A 27.218,B 90.000,C 0.000} C_DIS
LIN {X -256.740,Y -134.849,Z 139.091,A 27.710,B 90.000,C 0.000} C_DIS
LIN {X -255.573,Y -137.047,Z 139.327,A 28.202,B 90.000,C 0.000} C_DIS
LIN {X -254.390,Y -139.233,Z 139.595,A 28.693,B 90.000,C 0.000} C_DIS
LIN {X -253.189,Y -141.403,Z 139.908,A 29.183,B 90.000,C 0.000} C_DIS
LIN {X -251.974,Y -143.557,Z 140.268,A 29.671,B 90.000,C 0.000} C_DIS
LIN {X -250.745,Y -145.694,Z 140.682,A 30.158,B 90.000,C 0.000} C_DIS
LIN {X -250.240,Y -146.561,Z 140.867,A 30.357,B 90.000,C 0.000} C_DIS
LIN {X -248.514,Y -145.550,Z 140.867,A 30.357,B 90.000,C 0.000} C_DIS
WAIT SEC 0.1
RET=EKI_SetBool("oxy","torchState",FALSE)
RET = EKI_Send("oxy","torchState")
LIN {X -232.982,Y -136.453,Z 140.867,A 30.357,B 90.000,C 0.000} C_DIS
LIN {X -218.765,Y -158.247,Z 147.933,A 35.881,B 90.000,C 0.000} C_DIS
LIN {X -233.349,Y -168.797,Z 147.933,A 35.881,B 90.000,C 0.000} C_DIS
LIN {X -234.969,Y -169.969,Z 147.933,A 35.881,B 90.000,C 0.000} C_DIS
WAIT SEC 1.75
RET=EKI_SetBool("oxy","torchState",TRUE)
RET = EKI_Send("oxy","torchState")
LIN {X -233.526,Y -171.945,Z 148.444,A 36.364,B 90.000,C 0.000} C_DIS
LIN {X -232.062,Y -173.916,Z 148.915,A 36.849,B 90.000,C 0.000} C_DIS
LIN {X -230.578,Y -175.878,Z 149.356,A 37.335,B 90.000,C 0.000} C_DIS
LIN {X -229.075,Y -177.830,Z 149.780,A 37.822,B 90.000,C 0.000} C_DIS
LIN {X -227.555,Y -179.770,Z 150.198,A 38.309,B 90.000,C 0.000} C_DIS
LIN {X -226.020,Y -181.698,Z 150.618,A 38.796,B 90.000,C 0.000} C_DIS
LIN {X -224.471,Y -183.610,Z 151.053,A 39.282,B 90.000,C 0.000} C_DIS
LIN {X -222.907,Y -185.505,Z 151.514,A 39.768,B 90.000,C 0.000} C_DIS
LIN {X -221.332,Y -187.381,Z 152.014,A 40.251,B 90.000,C 0.000} C_DIS
LIN {X -219.748,Y -189.236,Z 152.560,A 40.733,B 90.000,C 0.000} C_DIS
LIN {X -218.158,Y -191.067,Z 153.166,A 41.213,B 90.000,C 0.000} C_DIS
LIN {X -217.516,Y -191.798,Z 153.429,A 41.405,B 90.000,C 0.000} C_DIS
LIN {X -216.016,Y -190.476,Z 153.429,A 41.405,B 90.000,C 0.000} C_DIS
WAIT SEC 0.1
RET=EKI_SetBool("oxy","torchState",FALSE)
RET = EKI_Send("oxy","torchState")
LIN {X -202.515,Y -178.571,Z 153.429,A 41.405,B 90.000,C 0.000} C_DIS
LIN {X -217.286,Y -160.271,Z 172.416,A 36.413,B 90.000,C 0.000} C_DIS
LIN {X -231.772,Y -170.956,Z 172.416,A 36.413,B 90.000,C 0.000} C_DIS
LIN {X -233.381,Y -172.143,Z 172.416,A 36.413,B 90.000,C 0.000} C_DIS
WAIT SEC 1.75
RET=EKI_SetBool("oxy","torchState",TRUE)
RET = EKI_Send("oxy","torchState")
LIN {X -234.389,Y -170.768,Z 170.588,A 36.076,B 90.000,C 0.000} C_DIS
LIN {X -235.617,Y -169.070,Z 169.224,A 35.662,B 90.000,C 0.000} C_DIS
LIN {X -236.992,Y -167.137,Z 168.435,A 35.193,B 90.000,C 0.000} C_DIS
LIN {X -238.422,Y -165.091,Z 168.304,A 34.700,B 90.000,C 0.000} C_DIS
LIN {X -239.803,Y -163.078,Z 168.837,A 34.218,B 90.000,C 0.000} C_DIS
LIN {X -241.045,Y -161.237,Z 169.986,A 33.779,B 90.000,C 0.000} C_DIS
LIN {X -242.079,Y -159.680,Z 171.646,A 33.410,B 90.000,C 0.000} C_DIS
LIN {X -242.865,Y -158.482,Z 173.694,A 33.126,B 90.000,C 0.000} C_DIS
LIN {X -243.384,Y -157.684,Z 176.005,A 32.939,B 90.000,C 0.000} C_DIS
LIN {X -243.626,Y -157.310,Z 178.465,A 32.850,B 90.000,C 0.000} C_DIS
LIN {X -243.587,Y -157.370,Z 180.964,A 32.865,B 90.000,C 0.000} C_DIS
LIN {X -243.269,Y -157.861,Z 183.394,A 32.980,B 90.000,C 0.000} C_DIS
LIN {X -242.677,Y -158.771,Z 185.646,A 33.195,B 90.000,C 0.000} C_DIS
LIN {X -241.819,Y -160.073,Z 187.600,A 33.503,B 90.000,C 0.000} C_DIS
LIN {X -240.724,Y -161.716,Z 189.132,A 33.893,B 90.000,C 0.000} C_DIS
LIN {X -239.436,Y -163.617,Z 190.121,A 34.346,B 90.000,C 0.000} C_DIS
LIN {X -238.031,Y -165.654,Z 190.476,A 34.835,B 90.000,C 0.000} C_DIS
LIN {X -236.606,Y -167.683,Z 190.159,A 35.325,B 90.000,C 0.000} C_DIS
LIN {X -235.263,Y -169.562,Z 189.204,A 35.782,B 90.000,C 0.000} C_DIS
LIN {X -234.090,Y -171.178,Z 187.700,A 36.176,B 90.000,C 0.000} C_DIS
LIN {X -233.151,Y -172.454,Z 185.766,A 36.489,B 90.000,C 0.000} C_DIS
LIN {X -232.487,Y -173.349,Z 183.529,A 36.709,B 90.000,C 0.000} C_DIS
LIN {X -232.119,Y -173.841,Z 181.106,A 36.831,B 90.000,C 0.000} C_DIS
LIN {X -232.060,Y -173.920,Z 178.608,A 36.850,B 90.000,C 0.000} C_DIS
LIN {X -232.308,Y -173.588,Z 176.143,A 36.768,B 90.000,C 0.000} C_DIS
LIN {X -232.859,Y -172.849,Z 173.820,A 36.586,B 90.000,C 0.000} C_DIS
LIN {X -233.381,Y -172.143,Z 172.416,A 36.413,B 90.000,C 0.000} C_DIS
LIN {X -231.772,Y -170.956,Z 172.416,A 36.413,B 90.000,C 0.000} C_DIS
WAIT SEC 0.1
RET=EKI_SetBool("oxy","torchState",FALSE)
RET = EKI_Send("oxy","torchState")
LIN {X -217.286,Y -160.271,Z 172.416,A 36.413,B 90.000,C 0.000} C_DIS
LIN {X -220.942,Y -155.192,Z 210.280,A 35.085,B 90.000,C 0.000} C_DIS
LIN {X -235.672,Y -165.538,Z 210.280,A 35.085,B 90.000,C 0.000} C_DIS
LIN {X -237.308,Y -166.688,Z 210.280,A 35.085,B 90.000,C 0.000} C_DIS
WAIT SEC 1.75
RET=EKI_SetBool("oxy","torchState",TRUE)
RET = EKI_Send("oxy","torchState")
LIN {X -235.901,Y -168.673,Z 209.708,A 35.565,B 90.000,C 0.000} C_DIS
LIN {X -234.488,Y -170.631,Z 209.061,A 36.042,B 90.000,C 0.000} C_DIS
LIN {X -233.071,Y -172.562,Z 208.346,A 36.516,B 90.000,C 0.000} C_DIS
LIN {X -231.649,Y -174.466,Z 207.571,A 36.985,B 90.000,C 0.000} C_DIS
LIN {X -230.222,Y -176.345,Z 206.745,A 37.451,B 90.000,C 0.000} C_DIS
LIN {X -228.790,Y -178.200,Z 205.877,A 37.914,B 90.000,C 0.000} C_DIS
LIN {X -227.350,Y -180.031,Z 204.970,A 38.375,B 90.000,C 0.000} C_DIS
LIN {X -225.903,Y -181.844,Z 204.037,A 38.833,B 90.000,C 0.000} C_DIS
LIN {X -224.448,Y -183.639,Z 203.084,A 39.289,B 90.000,C 0.000} C_DIS
LIN {X -222.980,Y -185.417,Z 202.117,A 39.745,B 90.000,C 0.000} C_DIS
LIN {X -221.498,Y -187.179,Z 201.145,A 40.200,B 90.000,C 0.000} C_DIS
LIN {X -220.006,Y -188.935,Z 200.175,A 40.655,B 90.000,C 0.000} C_DIS
LIN {X -218.497,Y -190.680,Z 199.212,A 41.111,B 90.000,C 0.000} C_DIS
LIN {X -216.969,Y -192.417,Z 198.267,A 41.568,B 90.000,C 0.000} C_DIS
LIN {X -215.419,Y -194.149,Z 197.346,A 42.027,B 90.000,C 0.000} C_DIS
LIN {X -213.850,Y -195.878,Z 196.454,A 42.488,B 90.000,C 0.000} C_DIS
LIN {X -213.799,Y -195.933,Z 196.426,A 42.503,B 90.000,C 0.000} C_DIS
LIN {X -212.325,Y -194.582,Z 196.426,A 42.503,B 90.000,C 0.000} C_DIS
WAIT SEC 0.1
RET=EKI_SetBool("oxy","torchState",FALSE)
RET = EKI_Send("oxy","torchState")
LIN {X -199.055,Y -182.421,Z 196.426,A 42.503,B 90.000,C 0.000} C_DIS
LIN {X -183.751,Y -197.827,Z 191.864,A 47.113,B 90.000,C 0.000} C_DIS
LIN {X -196.001,Y -211.015,Z 191.864,A 47.113,B 90.000,C 0.000} C_DIS
LIN {X -197.362,Y -212.481,Z 191.864,A 47.113,B 90.000,C 0.000} C_DIS
WAIT SEC 1.75
RET=EKI_SetBool("oxy","torchState",TRUE)
RET = EKI_Send("oxy","torchState")
LIN {X -195.530,Y -214.168,Z 192.079,A 47.605,B 90.000,C 0.000} C_DIS
LIN {X -193.698,Y -215.826,Z 192.451,A 48.093,B 90.000,C 0.000} C_DIS
LIN {X -191.871,Y -217.452,Z 192.968,A 48.576,B 90.000,C 0.000} C_DIS
LIN {X -190.054,Y -219.042,Z 193.615,A 49.053,B 90.000,C 0.000} C_DIS
LIN {X -188.249,Y -220.595,Z 194.378,A 49.523,B 90.000,C 0.000} C_DIS
LIN {X -186.459,Y -222.110,Z 195.244,A 49.987,B 90.000,C 0.000} C_DIS
LIN {X -184.683,Y -223.589,Z 196.195,A 50.444,B 90.000,C 0.000} C_DIS
LIN {X -182.919,Y -225.035,Z 197.219,A 50.894,B 90.000,C 0.000} C_DIS
LIN {X -181.166,Y -226.448,Z 198.304,A 51.339,B 90.000,C 0.000} C_DIS
LIN {X -179.421,Y -227.833,Z 199.438,A 51.779,B 90.000,C 0.000} C_DIS
LIN {X -177.681,Y -229.192,Z 200.610,A 52.215,B 90.000,C 0.000} C_DIS
LIN {X -175.942,Y -230.529,Z 201.808,A 52.649,B 90.000,C 0.000} C_DIS
LIN {X -174.200,Y -231.848,Z 203.023,A 53.080,B 90.000,C 0.000} C_DIS
LIN {X -173.006,Y -232.742,Z 203.858,A 53.375,B 90.000,C 0.000} C_DIS
LIN {X -171.813,Y -231.137,Z 203.858,A 53.375,B 90.000,C 0.000} C_DIS
WAIT SEC 0.1
RET=EKI_SetBool("oxy","torchState",FALSE)
RET = EKI_Send("oxy","torchState")
LIN {X -161.074,Y -216.691,Z 203.858,A 53.375,B 90.000,C 0.000} C_DIS
LIN {X -144.956,Y -227.789,Z 182.478,A 57.529,B 90.000,C 0.000} C_DIS
LIN {X -154.620,Y -242.975,Z 182.478,A 57.529,B 90.000,C 0.000} C_DIS
LIN {X -155.694,Y -244.662,Z 182.478,A 57.529,B 90.000,C 0.000} C_DIS
WAIT SEC 1.75
RET=EKI_SetBool("oxy","torchState",TRUE)
RET = EKI_Send("oxy","torchState")
LIN {X -157.782,Y -243.320,Z 182.182,A 57.038,B 90.000,C 0.000} C_DIS
LIN {X -159.867,Y -241.955,Z 181.991,A 56.546,B 90.000,C 0.000} C_DIS
LIN {X -161.942,Y -240.571,Z 181.822,A 56.053,B 90.000,C 0.000} C_DIS
LIN {X -164.002,Y -239.172,Z 181.601,A 55.561,B 90.000,C 0.000} C_DIS
LIN {X -166.041,Y -237.761,Z 181.284,A 55.071,B 90.000,C 0.000} C_DIS
LIN {X -168.055,Y -236.341,Z 180.867,A 54.585,B 90.000,C 0.000} C_DIS
LIN {X -170.044,Y -234.914,Z 180.361,A 54.101,B 90.000,C 0.000} C_DIS
LIN {X -172.006,Y -233.482,Z 179.772,A 53.621,B 90.000,C 0.000} C_DIS
LIN {X -173.940,Y -232.045,Z 179.104,A 53.145,B 90.000,C 0.000} C_DIS
LIN {X -175.844,Y -230.605,Z 178.365,A 52.673,B 90.000,C 0.000} C_DIS
LIN {X -177.721,Y -229.162,Z 177.563,A 52.205,B 90.000,C 0.000} C_DIS
LIN {X -179.570,Y -227.716,Z 176.702,A 51.742,B 90.000,C 0.000} C_DIS
LIN {X -181.391,Y -226.268,Z 175.789,A 51.282,B 90.000,C 0.000} C_DIS
LIN {X -183.186,Y -224.817,Z 174.828,A 50.826,B 90.000,C 0.000} C_DIS
LIN {X -184.956,Y -223.363,Z 173.829,A 50.373,B 90.000,C 0.000} C_DIS
LIN {X -186.702,Y -221.904,Z 172.793,A 49.924,B 90.000,C 0.000} C_DIS
LIN {X -188.428,Y -220.442,Z 171.728,A 49.477,B 90.000,C 0.000} C_DIS
LIN {X -190.132,Y -218.974,Z 170.638,A 49.033,B 90.000,C 0.000} C_DIS
LIN {X -191.817,Y -217.499,Z 169.527,A 48.590,B 90.000,C 0.000} C_DIS
LIN {X -192.303,Y -217.070,Z 169.202,A 48.462,B 90.000,C 0.000} C_DIS
LIN {X -190.977,Y -215.573,Z 169.202,A 48.462,B 90.000,C 0.000} C_DIS
WAIT SEC 0.1
RET=EKI_SetBool("oxy","torchState",FALSE)
RET = EKI_Send("oxy","torchState")
LIN {X -179.041,Y -202.100,Z 169.202,A 48.462,B 90.000,C 0.000} C_DIS
LIN {X -176.775,Y -204.085,Z 132.741,A 49.101,B 90.000,C 0.000} C_DIS
LIN {X -188.560,Y -217.690,Z 132.741,A 49.101,B 90.000,C 0.000} C_DIS
LIN {X -189.870,Y -219.202,Z 132.741,A 49.101,B 90.000,C 0.000} C_DIS
WAIT SEC 1.75
RET=EKI_SetBool("oxy","torchState",TRUE)
RET = EKI_Send("oxy","torchState")
LIN {X -191.663,Y -217.633,Z 131.986,A 48.631,B 90.000,C 0.000} C_DIS
LIN {X -193.447,Y -216.048,Z 131.241,A 48.159,B 90.000,C 0.000} C_DIS
LIN {X -195.221,Y -214.447,Z 130.509,A 47.687,B 90.000,C 0.000} C_DIS
LIN {X -196.986,Y -212.827,Z 129.793,A 47.214,B 90.000,C 0.000} C_DIS
LIN {X -198.740,Y -211.190,Z 129.093,A 46.740,B 90.000,C 0.000} C_DIS
LIN {X -200.485,Y -209.535,Z 128.411,A 46.264,B 90.000,C 0.000} C_DIS
LIN {X -202.220,Y -207.863,Z 127.748,A 45.788,B 90.000,C 0.000} C_DIS
LIN {X -203.945,Y -206.170,Z 127.109,A 45.311,B 90.000,C 0.000} C_DIS
LIN {X -205.659,Y -204.459,Z 126.492,A 44.832,B 90.000,C 0.000} C_DIS
LIN {X -207.364,Y -202.730,Z 125.898,A 44.353,B 90.000,C 0.000} C_DIS
LIN {X -209.059,Y -200.982,Z 125.331,A 43.872,B 90.000,C 0.000} C_DIS
LIN {X -210.743,Y -199.215,Z 124.793,A 43.389,B 90.000,C 0.000} C_DIS
LIN {X -212.417,Y -197.430,Z 124.282,A 42.906,B 90.000,C 0.000} C_DIS
LIN {X -214.080,Y -195.625,Z 123.805,A 42.421,B 90.000,C 0.000} C_DIS
LIN {X -215.731,Y -193.803,Z 123.359,A 41.935,B 90.000,C 0.000} C_DIS
LIN {X -217.371,Y -191.961,Z 122.949,A 41.448,B 90.000,C 0.000} C_DIS
LIN {X -219.000,Y -190.102,Z 122.574,A 40.960,B 90.000,C 0.000} C_DIS
LIN {X -220.615,Y -188.224,Z 122.238,A 40.470,B 90.000,C 0.000} C_DIS
LIN {X -222.218,Y -186.330,Z 121.940,A 39.980,B 90.000,C 0.000} C_DIS
LIN {X -223.807,Y -184.417,Z 121.686,A 39.489,B 90.000,C 0.000} C_DIS
LIN {X -224.128,Y -184.029,Z 121.638,A 39.389,B 90.000,C 0.000} C_DIS
LIN {X -222.582,Y -182.760,Z 121.638,A 39.389,B 90.000,C 0.000} C_DIS
WAIT SEC 0.1
RET=EKI_SetBool("oxy","torchState",FALSE)
RET = EKI_Send("oxy","torchState")
LIN {X -208.671,Y -171.337,Z 121.638,A 39.389,B 90.000,C 0.000} C_DIS
LIN {X -221.861,Y -153.876,Z 120.528,A 34.744,B 90.000,C 0.000} C_DIS
LIN {X -236.652,Y -164.134,Z 120.528,A 34.744,B 90.000,C 0.000} C_DIS
LIN {X -238.295,Y -165.274,Z 120.528,A 34.744,B 90.000,C 0.000} C_DIS
WAIT SEC 1.75
RET=EKI_SetBool("oxy","torchState",TRUE)
RET = EKI_Send("oxy","torchState")
LIN {X -239.707,Y -163.215,Z 120.409,A 34.251,B 90.000,C 0.000} C_DIS
LIN {X -241.103,Y -161.146,Z 120.274,A 33.757,B 90.000,C 0.000} C_DIS
LIN {X -242.481,Y -159.066,Z 120.120,A 33.265,B 90.000,C 0.000} C_DIS
LIN {X -243.840,Y -156.975,Z 119.948,A 32.772,B 90.000,C 0.000} C_DIS
LIN {X -245.181,Y -154.874,Z 119.756,A 32.279,B 90.000,C 0.000} C_DIS
LIN {X -246.502,Y -152.762,Z 119.545,A 31.787,B 90.000,C 0.000} C_DIS
LIN {X -247.804,Y -150.641,Z 119.314,A 31.296,B 90.000,C 0.000} C_DIS
LIN {X -249.086,Y -148.510,Z 119.063,A 30.804,B 90.000,C 0.000} C_DIS
LIN {X -250.349,Y -146.370,Z 118.793,A 30.313,B 90.000,C 0.000} C_DIS
LIN {X -251.593,Y -144.221,Z 118.503,A 29.823,B 90.000,C 0.000} C_DIS
LIN {X -252.818,Y -142.064,Z 118.193,A 29.333,B 90.000,C 0.000} C_DIS
LIN {X -254.023,Y -139.899,Z 117.864,A 28.843,B 90.000,C 0.000} C_DIS
LIN {X -255.208,Y -137.726,Z 117.514,A 28.354,B 90.000,C 0.000} C_DIS
LIN {X -256.373,Y -135.546,Z 117.144,A 27.866,B 90.000,C 0.000} C_DIS
LIN {X -257.517,Y -133.358,Z 116.752,A 27.378,B 90.000,C 0.000} C_DIS
LIN {X -258.641,Y -131.163,Z 116.339,A 26.891,B 90.000,C 0.000} C_DIS
LIN {X -259.745,Y -128.963,Z 115.905,A 26.404,B 90.000,C 0.000} C_DIS
LIN {X -260.829,Y -126.757,Z 115.451,A 25.919,B 90.000,C 0.000} C_DIS
LIN {X -261.893,Y -124.545,Z 114.976,A 25.434,B 90.000,C 0.000} C_DIS
LIN {X -262.937,Y -122.329,Z 114.480,A 24.950,B 90.000,C 0.000} C_DIS
LIN {X -263.958,Y -120.107,Z 113.961,A 24.467,B 90.000,C 0.000} C_DIS
LIN {X -264.959,Y -117.881,Z 113.420,A 23.984,B 90.000,C 0.000} C_DIS
LIN {X -265.939,Y -115.652,Z 112.857,A 23.503,B 90.000,C 0.000} C_DIS
LIN {X -266.900,Y -113.419,Z 112.274,A 23.023,B 90.000,C 0.000} C_DIS
LIN {X -267.840,Y -111.183,Z 111.668,A 22.544,B 90.000,C 0.000} C_DIS
LIN {X -268.757,Y -108.945,Z 111.039,A 22.066,B 90.000,C 0.000} C_DIS
LIN {X -269.654,Y -106.704,Z 110.387,A 21.589,B 90.000,C 0.000} C_DIS
LIN {X -270.530,Y -104.462,Z 109.713,A 21.114,B 90.000,C 0.000} C_DIS
LIN {X -271.386,Y -102.219,Z 109.018,A 20.639,B 90.000,C 0.000} C_DIS
LIN {X -272.206,Y -100.020,Z 108.314,A 20.175,B 90.000,C 0.000} C_DIS
LIN {X -270.329,Y -99.330,Z 108.314,A 20.175,B 90.000,C 0.000} C_DIS
WAIT SEC 0.1
RET=EKI_SetBool("oxy","torchState",FALSE)
RET = EKI_Send("oxy","torchState")
LIN {X -253.433,Y -93.122,Z 108.314,A 20.175,B 90.000,C 0.000} C_DIS
LIN {X -251.129,Y -99.167,Z 69.422,A 21.548,B 90.000,C 0.000} C_DIS
LIN {X -267.871,Y -105.778,Z 69.422,A 21.548,B 90.000,C 0.000} C_DIS
LIN {X -269.732,Y -106.512,Z 69.422,A 21.548,B 90.000,C 0.000} C_DIS
WAIT SEC 1.75
RET=EKI_SetBool("oxy","torchState",TRUE)
RET = EKI_Send("oxy","torchState")
LIN {X -268.862,Y -108.689,Z 70.291,A 22.011,B 90.000,C 0.000} C_DIS
LIN {X -267.974,Y -110.856,Z 71.165,A 22.474,B 90.000,C 0.000} C_DIS
LIN {X -267.070,Y -113.019,Z 72.034,A 22.937,B 90.000,C 0.000} C_DIS
LIN {X -266.146,Y -115.179,Z 72.886,A 23.401,B 90.000,C 0.000} C_DIS
LIN {X -265.200,Y -117.341,Z 73.711,A 23.868,B 90.000,C 0.000} C_DIS
LIN {X -264.231,Y -119.507,Z 74.497,A 24.336,B 90.000,C 0.000} C_DIS
LIN {X -263.237,Y -121.679,Z 75.234,A 24.808,B 90.000,C 0.000} C_DIS
LIN {X -262.548,Y -123.161,Z 75.703,A 25.131,B 90.000,C 0.000} C_DIS
LIN {X -260.737,Y -122.312,Z 75.703,A 25.131,B 90.000,C 0.000} C_DIS
WAIT SEC 0.1
RET=EKI_SetBool("oxy","torchState",FALSE)
RET = EKI_Send("oxy","torchState")
LIN {X -244.441,Y -114.667,Z 75.703,A 25.131,B 90.000,C 0.000} C_DIS
LIN {X -240.717,Y -122.291,Z 50.578,A 26.932,B 90.000,C 0.000} C_DIS
LIN {X -256.765,Y -130.444,Z 50.578,A 26.932,B 90.000,C 0.000} C_DIS
LIN {X -258.548,Y -131.350,Z 50.578,A 26.932,B 90.000,C 0.000} C_DIS
WAIT SEC 1.75
RET=EKI_SetBool("oxy","torchState",TRUE)
RET = EKI_Send("oxy","torchState")
LIN {X -259.668,Y -129.121,Z 50.407,A 26.439,B 90.000,C 0.000} C_DIS
LIN {X -260.767,Y -126.886,Z 50.195,A 25.947,B 90.000,C 0.000} C_DIS
LIN {X -261.846,Y -124.645,Z 49.946,A 25.456,B 90.000,C 0.000} C_DIS
LIN {X -262.903,Y -122.399,Z 49.654,A 24.965,B 90.000,C 0.000} C_DIS
LIN {X -263.939,Y -120.148,Z 49.325,A 24.476,B 90.000,C 0.000} C_DIS
LIN {X -264.954,Y -117.894,Z 48.955,A 23.987,B 90.000,C 0.000} C_DIS
LIN {X -265.947,Y -115.636,Z 48.546,A 23.500,B 90.000,C 0.000} C_DIS
LIN {X -266.919,Y -113.377,Z 48.100,A 23.014,B 90.000,C 0.000} C_DIS
LIN {X -267.867,Y -111.116,Z 47.612,A 22.530,B 90.000,C 0.000} C_DIS
LIN {X -268.794,Y -108.855,Z 47.088,A 22.047,B 90.000,C 0.000} C_DIS
LIN {X -269.698,Y -106.594,Z 46.522,A 21.566,B 90.000,C 0.000} C_DIS
LIN {X -270.581,Y -104.334,Z 45.920,A 21.086,B 90.000,C 0.000} C_DIS
LIN {X -271.441,Y -102.076,Z 45.279,A 20.609,B 90.000,C 0.000} C_DIS
LIN {X -272.278,Y -99.821,Z 44.600,A 20.134,B 90.000,C 0.000} C_DIS
LIN {X -273.094,Y -97.569,Z 43.884,A 19.660,B 90.000,C 0.000} C_DIS
LIN {X -273.885,Y -95.322,Z 43.128,A 19.190,B 90.000,C 0.000} C_DIS
LIN {X -274.656,Y -93.080,Z 42.337,A 18.721,B 90.000,C 0.000} C_DIS
LIN {X -275.403,Y -90.844,Z 41.506,A 18.255,B 90.000,C 0.000} C_DIS
LIN {X -276.129,Y -88.614,Z 40.639,A 17.792,B 90.000,C 0.000} C_DIS
LIN {X -276.832,Y -86.392,Z 39.735,A 17.332,B 90.000,C 0.000} C_DIS
LIN {X -277.513,Y -84.179,Z 38.793,A 16.874,B 90.000,C 0.000} C_DIS
LIN {X -278.173,Y -81.975,Z 37.816,A 16.420,B 90.000,C 0.000} C_DIS
LIN {X -278.809,Y -79.782,Z 36.799,A 15.969,B 90.000,C 0.000} C_DIS
LIN {X -279.425,Y -77.599,Z 35.749,A 15.520,B 90.000,C 0.000} C_DIS
LIN {X -280.018,Y -75.428,Z 34.660,A 15.076,B 90.000,C 0.000} C_DIS
LIN {X -280.115,Y -75.070,Z 34.479,A 15.003,B 90.000,C 0.000} C_DIS
LIN {X -278.183,Y -74.552,Z 34.479,A 15.003,B 90.000,C 0.000} C_DIS
WAIT SEC 0.1
RET=EKI_SetBool("oxy","torchState",FALSE)
RET = EKI_Send("oxy","torchState")
LIN {X -260.797,Y -69.893,Z 34.479,A 15.003,B 90.000,C 0.000} C_DIS
LIN {X -266.530,Y -43.150,Z 86.108,A 9.196,B 90.000,C 0.000} C_DIS
LIN {X -284.298,Y -46.027,Z 86.108,A 9.196,B 90.000,C 0.000} C_DIS
LIN {X -286.273,Y -46.347,Z 86.108,A 9.196,B 90.000,C 0.000} C_DIS
WAIT SEC 1.75
RET=EKI_SetBool("oxy","torchState",TRUE)
RET = EKI_Send("oxy","torchState")
LIN {X -286.624,Y -44.106,Z 85.057,A 8.748,B 90.000,C 0.000} C_DIS
LIN {X -286.960,Y -41.863,Z 84.006,A 8.300,B 90.000,C 0.000} C_DIS
LIN {X -287.277,Y -39.616,Z 82.957,A 7.852,B 90.000,C 0.000} C_DIS
LIN {X -287.581,Y -37.367,Z 81.911,A 7.403,B 90.000,C 0.000} C_DIS
LIN {X -287.867,Y -35.111,Z 80.872,A 6.954,B 90.000,C 0.000} C_DIS
LIN {X -288.133,Y -32.848,Z 79.845,A 6.504,B 90.000,C 0.000} C_DIS
LIN {X -288.383,Y -30.577,Z 78.830,A 6.052,B 90.000,C 0.000} C_DIS
LIN {X -288.615,Y -28.296,Z 77.833,A 5.599,B 90.000,C 0.000} C_DIS
LIN {X -288.830,Y -26.006,Z 76.855,A 5.145,B 90.000,C 0.000} C_DIS
LIN {X -289.028,Y -23.705,Z 75.899,A 4.689,B 90.000,C 0.000} C_DIS
LIN {X -289.210,Y -21.392,Z 74.968,A 4.230,B 90.000,C 0.000} C_DIS
LIN {X -289.371,Y -19.066,Z 74.067,A 3.770,B 90.000,C 0.000} C_DIS
LIN {X -289.517,Y -16.728,Z 73.195,A 3.307,B 90.000,C 0.000} C_DIS
LIN {X -289.643,Y -14.375,Z 72.362,A 2.841,B 90.000,C 0.000} C_DIS
LIN {X -289.737,Y -12.345,Z 71.674,A 2.440,B 90.000,C 0.000} C_DIS
LIN {X -287.739,Y -12.260,Z 71.674,A 2.440,B 90.000,C 0.000} C_DIS
WAIT SEC 0.1
RET=EKI_SetBool("oxy","torchState",FALSE)
RET = EKI_Send("oxy","torchState")
LIN {X -269.755,Y -11.494,Z 71.674,A 2.440,B 90.000,C 0.000} C_DIS
LIN {X -269.988,Y 2.582,Z 45.084,A -0.548,B 90.000,C 0.000} C_DIS
LIN {X -287.987,Y 2.754,Z 45.084,A -0.548,B 90.000,C 0.000} C_DIS
LIN {X -289.987,Y 2.773,Z 45.084,A -0.548,B 90.000,C 0.000} C_DIS
WAIT SEC 1.75
RET=EKI_SetBool("oxy","torchState",TRUE)
RET = EKI_Send("oxy","torchState")
LIN {X -289.948,Y 5.261,Z 44.845,A -1.039,B 90.000,C 0.000} C_DIS
LIN {X -289.893,Y 7.749,Z 44.615,A -1.531,B 90.000,C 0.000} C_DIS
LIN {X -289.818,Y 10.238,Z 44.393,A -2.023,B 90.000,C 0.000} C_DIS
LIN {X -289.719,Y 12.727,Z 44.183,A -2.515,B 90.000,C 0.000} C_DIS
LIN {X -289.597,Y 15.216,Z 43.984,A -3.008,B 90.000,C 0.000} C_DIS
LIN {X -289.455,Y 17.704,Z 43.795,A -3.500,B 90.000,C 0.000} C_DIS
LIN {X -289.293,Y 20.192,Z 43.615,A -3.993,B 90.000,C 0.000} C_DIS
LIN {X -289.110,Y 22.679,Z 43.445,A -4.485,B 90.000,C 0.000} C_DIS
LIN {X -288.905,Y 25.165,Z 43.286,A -4.978,B 90.000,C 0.000} C_DIS
LIN {X -288.675,Y 27.650,Z 43.138,A -5.471,B 90.000,C 0.000} C_DIS
LIN {X -288.426,Y 30.134,Z 42.999,A -5.964,B 90.000,C 0.000} C_DIS
LIN {X -288.157,Y 32.615,Z 42.870,A -6.458,B 90.000,C 0.000} C_DIS
LIN {X -287.867,Y 35.095,Z 42.751,A -6.951,B 90.000,C 0.000} C_DIS
LIN {X -287.554,Y 37.573,Z 42.643,A -7.444,B 90.000,C 0.000} C_DIS
LIN {X -287.218,Y 40.048,Z 42.546,A -7.938,B 90.000,C 0.000} C_DIS
LIN {X -286.862,Y 42.521,Z 42.458,A -8.431,B 90.000,C 0.000} C_DIS
LIN {X -286.485,Y 44.991,Z 42.380,A -8.925,B 90.000,C 0.000} C_DIS
LIN {X -286.089,Y 47.458,Z 42.312,A -9.419,B 90.000,C 0.000} C_DIS
LIN {X -285.669,Y 49.922,Z 42.255,A -9.913,B 90.000,C 0.000} C_DIS
LIN {X -285.226,Y 52.381,Z 42.208,A -10.406,B 90.000,C 0.000} C_DIS
LIN {X -284.764,Y 54.838,Z 42.172,A -10.900,B 90.000,C 0.000} C_DIS
LIN {X -284.281,Y 57.290,Z 42.145,A -11.394,B 90.000,C 0.000} C_DIS
LIN {X -283.779,Y 59.739,Z 42.128,A -11.888,B 90.000,C 0.000} C_DIS
LIN {X -283.253,Y 62.183,Z 42.122,A -12.382,B 90.000,C 0.000} C_DIS
LIN {X -282.705,Y 64.621,Z 42.126,A -12.876,B 90.000,C 0.000} C_DIS
LIN {X -282.137,Y 67.056,Z 42.141,A -13.369,B 90.000,C 0.000} C_DIS
LIN {X -281.549,Y 69.485,Z 42.165,A -13.863,B 90.000,C 0.000} C_DIS
LIN {X -280.942,Y 71.910,Z 42.199,A -14.357,B 90.000,C 0.000} C_DIS
LIN {X -280.311,Y 74.328,Z 42.244,A -14.851,B 90.000,C 0.000} C_DIS
LIN {X -280.215,Y 74.697,Z 42.251,A -14.926,B 90.000,C 0.000} C_DIS
LIN {X -279.573,Y 77.063,Z 41.761,A -15.411,B 90.000,C 0.000} C_DIS
LIN {X -278.908,Y 79.436,Z 41.343,A -15.898,B 90.000,C 0.000} C_DIS
LIN {X -278.220,Y 81.814,Z 40.998,A -16.387,B 90.000,C 0.000} C_DIS
LIN {X -277.508,Y 84.195,Z 40.725,A -16.878,B 90.000,C 0.000} C_DIS
LIN {X -277.037,Y 85.736,Z 40.585,A -17.196,B 90.000,C 0.000} C_DIS
LIN {X -275.126,Y 85.145,Z 40.585,A -17.196,B 90.000,C 0.000} C_DIS
WAIT SEC 0.1
RET=EKI_SetBool("oxy","torchState",FALSE)
RET = EKI_Send("oxy","torchState")
LIN {X -257.931,Y 79.823,Z 40.585,A -17.196,B 90.000,C 0.000} C_DIS
LIN {X -265.163,Y 50.880,Z 58.350,A -10.862,B 90.000,C 0.000} C_DIS
LIN {X -282.840,Y 54.271,Z 58.350,A -10.862,B 90.000,C 0.000} C_DIS
LIN {X -284.804,Y 54.648,Z 58.350,A -10.862,B 90.000,C 0.000} C_DIS
WAIT SEC 1.75
RET=EKI_SetBool("oxy","torchState",TRUE)
RET = EKI_Send("oxy","torchState")
LIN {X -285.260,Y 52.211,Z 58.669,A -10.372,B 90.000,C 0.000} C_DIS
LIN {X -285.695,Y 49.774,Z 59.013,A -9.883,B 90.000,C 0.000} C_DIS
LIN {X -286.109,Y 47.336,Z 59.379,A -9.394,B 90.000,C 0.000} C_DIS
LIN {X -286.502,Y 44.898,Z 59.763,A -8.906,B 90.000,C 0.000} C_DIS
LIN {X -286.874,Y 42.458,Z 60.162,A -8.419,B 90.000,C 0.000} C_DIS
LIN {X -287.222,Y 40.017,Z 60.572,A -7.932,B 90.000,C 0.000} C_DIS
LIN {X -287.549,Y 37.574,Z 60.988,A -7.445,B 90.000,C 0.000} C_DIS
LIN {X -287.862,Y 35.129,Z 61.407,A -6.958,B 90.000,C 0.000} C_DIS
LIN {X -288.055,Y 33.529,Z 61.681,A -6.639,B 90.000,C 0.000} C_DIS
LIN {X -286.069,Y 33.297,Z 61.681,A -6.639,B 90.000,C 0.000} C_DIS
WAIT SEC 0.1
RET=EKI_SetBool("oxy","torchState",FALSE)
RET = EKI_Send("oxy","torchState")
LIN {X -268.189,Y 31.216,Z 61.681,A -6.639,B 90.000,C 0.000} C_DIS
LIN {X -268.352,Y 29.785,Z 134.101,A -6.333,B 90.000,C 0.000} C_DIS
LIN {X -286.242,Y 31.770,Z 134.101,A -6.333,B 90.000,C 0.000} C_DIS
LIN {X -288.230,Y 31.991,Z 134.101,A -6.333,B 90.000,C 0.000} C_DIS
WAIT SEC 1.75
RET=EKI_SetBool("oxy","torchState",TRUE)
RET = EKI_Send("oxy","torchState")
LIN {X -288.494,Y 29.506,Z 134.152,A -5.840,B 90.000,C 0.000} C_DIS
LIN {X -288.737,Y 27.018,Z 134.179,A -5.346,B 90.000,C 0.000} C_DIS
LIN {X -288.960,Y 24.528,Z 134.184,A -4.852,B 90.000,C 0.000} C_DIS
LIN {X -289.160,Y 22.037,Z 134.170,A -4.358,B 90.000,C 0.000} C_DIS
LIN {X -289.338,Y 19.543,Z 134.143,A -3.864,B 90.000,C 0.000} C_DIS
LIN {X -289.493,Y 17.049,Z 134.106,A -3.370,B 90.000,C 0.000} C_DIS
LIN {X -289.631,Y 14.553,Z 134.066,A -2.877,B 90.000,C 0.000} C_DIS
LIN {X -289.748,Y 12.056,Z 134.025,A -2.383,B 90.000,C 0.000} C_DIS
LIN {X -289.841,Y 9.559,Z 133.983,A -1.889,B 90.000,C 0.000} C_DIS
LIN {X -289.913,Y 7.060,Z 133.950,A -1.395,B 90.000,C 0.000} C_DIS
LIN {X -289.964,Y 4.561,Z 133.929,A -0.901,B 90.000,C 0.000} C_DIS
LIN {X -289.993,Y 2.062,Z 133.923,A -0.407,B 90.000,C 0.000} C_DIS
LIN {X -289.999,Y -0.438,Z 133.937,A 0.087,B 90.000,C 0.000} C_DIS
LIN {X -289.984,Y -2.937,Z 133.976,A 0.580,B 90.000,C 0.000} C_DIS
LIN {X -289.948,Y -5.436,Z 134.042,A 1.074,B 90.000,C 0.000} C_DIS
LIN {X -289.891,Y -7.933,Z 134.140,A 1.568,B 90.000,C 0.000} C_DIS
LIN {X -289.812,Y -10.428,Z 134.277,A 2.061,B 90.000,C 0.000} C_DIS
LIN {X -289.711,Y -12.919,Z 134.454,A 2.553,B 90.000,C 0.000} C_DIS
LIN {X -289.590,Y -15.406,Z 134.675,A 3.045,B 90.000,C 0.000} C_DIS
LIN {X -289.447,Y -17.887,Z 134.949,A 3.536,B 90.000,C 0.000} C_DIS
LIN {X -289.284,Y -20.359,Z 135.278,A 4.026,B 90.000,C 0.000} C_DIS
LIN {X -289.100,Y -22.822,Z 135.664,A 4.514,B 90.000,C 0.000} C_DIS
LIN {X -288.896,Y -25.273,Z 136.112,A 5.000,B 90.000,C 0.000} C_DIS
LIN {X -288.673,Y -27.709,Z 136.627,A 5.483,B 90.000,C 0.000} C_DIS
LIN {X -288.454,Y -29.901,Z 137.151,A 5.918,B 90.000,C 0.000} C_DIS
LIN {X -286.465,Y -29.694,Z 137.151,A 5.918,B 90.000,C 0.000} C_DIS
WAIT SEC 0.1
RET=EKI_SetBool("oxy","torchState",FALSE)
RET = EKI_Send("oxy","torchState")
LIN {X -268.561,Y -27.839,Z 137.151,A 5.918,B 90.000,C 0.000} C_DIS
LIN {X -267.760,Y -34.706,Z 178.909,A 7.385,B 90.000,C 0.000} C_DIS
LIN {X -285.611,Y -37.020,Z 178.909,A 7.385,B 90.000,C 0.000} C_DIS
LIN {X -287.594,Y -37.277,Z 178.909,A 7.385,B 90.000,C 0.000} C_DIS
WAIT SEC 1.75
RET=EKI_SetBool("oxy","torchState",TRUE)
RET = EKI_Send("oxy","torchState")
LIN {X -287.305,Y -39.438,Z 180.131,A 7.816,B 90.000,C 0.000} C_DIS
LIN {X -287.003,Y -41.583,Z 181.378,A 8.244,B 90.000,C 0.000} C_DIS
LIN {X -286.686,Y -43.713,Z 182.648,A 8.669,B 90.000,C 0.000} C_DIS
LIN {X -286.355,Y -45.828,Z 183.939,A 9.092,B 90.000,C 0.000} C_DIS
LIN {X -286.010,Y -47.931,Z 185.245,A 9.513,B 90.000,C 0.000} C_DIS
LIN {X -285.651,Y -50.024,Z 186.564,A 9.933,B 90.000,C 0.000} C_DIS
LIN {X -285.278,Y -52.109,Z 187.891,A 10.352,B 90.000,C 0.000} C_DIS
LIN {X -284.890,Y -54.188,Z 189.224,A 10.769,B 90.000,C 0.000} C_DIS
LIN {X -284.486,Y -56.262,Z 190.560,A 11.187,B 90.000,C 0.000} C_DIS
LIN {X -284.070,Y -58.334,Z 191.894,A 11.604,B 90.000,C 0.000} C_DIS
LIN {X -283.639,Y -60.406,Z 193.225,A 12.022,B 90.000,C 0.000} C_DIS
LIN {X -283.189,Y -62.478,Z 194.548,A 12.442,B 90.000,C 0.000} C_DIS
LIN {X -282.723,Y -64.555,Z 195.860,A 12.862,B 90.000,C 0.000} C_DIS
LIN {X -282.239,Y -66.636,Z 197.156,A 13.284,B 90.000,C 0.000} C_DIS
LIN {X -281.738,Y -68.725,Z 198.435,A 13.709,B 90.000,C 0.000} C_DIS
LIN {X -281.218,Y -70.821,Z 199.693,A 14.135,B 90.000,C 0.000} C_DIS
LIN {X -281.023,Y -71.596,Z 200.152,A 14.293,B 90.000,C 0.000} C_DIS
LIN {X -279.085,Y -71.102,Z 200.152,A 14.293,B 90.000,C 0.000} C_DIS
WAIT SEC 0.1
RET=EKI_SetBool("oxy","torchState",FALSE)
RET = EKI_Send("oxy","torchState")
LIN {X -261.642,Y -66.658,Z 200.152,A 14.293,B 90.000,C 0.000} C_DIS
LIN {X -251.976,Y -96.995,Z 216.157,A 21.053,B 90.000,C 0.000} C_DIS
LIN {X -268.775,Y -103.461,Z 216.157,A 21.053,B 90.000,C 0.000} C_DIS
LIN {X -270.641,Y -104.179,Z 216.157,A 21.053,B 90.000,C 0.000} C_DIS
WAIT SEC 1.75
RET=EKI_SetBool("oxy","torchState",TRUE)
RET = EKI_Send("oxy","torchState")
LIN {X -269.792,Y -106.354,Z 217.050,A 21.515,B 90.000,C 0.000} C_DIS
LIN {X -268.925,Y -108.530,Z 217.923,A 21.978,B 90.000,C 0.000} C_DIS
LIN {X -268.036,Y -110.707,Z 218.771,A 22.442,B 90.000,C 0.000} C_DIS
LIN {X -267.125,Y -112.887,Z 219.587,A 22.909,B 90.000,C 0.000} C_DIS
LIN {X -266.193,Y -115.070,Z 220.372,A 23.378,B 90.000,C 0.000} C_DIS
LIN {X -265.237,Y -117.256,Z 221.116,A 23.849,B 90.000,C 0.000} C_DIS
LIN {X -264.258,Y -119.446,Z 221.818,A 24.323,B 90.000,C 0.000} C_DIS
LIN {X -263.255,Y -121.641,Z 222.474,A 24.800,B 90.000,C 0.000} C_DIS
LIN {X -262.229,Y -123.839,Z 223.077,A 25.279,B 90.000,C 0.000} C_DIS
LIN {X -261.178,Y -126.040,Z 223.622,A 25.761,B 90.000,C 0.000} C_DIS
LIN {X -260.102,Y -128.244,Z 224.106,A 26.246,B 90.000,C 0.000} C_DIS
LIN {X -259.003,Y -130.450,Z 224.524,A 26.733,B 90.000,C 0.000} C_DIS
LIN {X -257.880,Y -132.657,Z 224.869,A 27.222,B 90.000,C 0.000} C_DIS
LIN {X -256.890,Y -134.564,Z 225.108,A 27.646,B 90.000,C 0.000} C_DIS
LIN {X -255.119,Y -133.636,Z 225.108,A 27.646,B 90.000,C 0.000} C_DIS
WAIT SEC 0.1
RET=EKI_SetBool("oxy","torchState",FALSE)
RET = EKI_Send("oxy","torchState")
LIN {X -239.174,Y -125.283,Z 225.108,A 27.646,B 90.000,C 0.000} C_DIS
LIN {X -233.387,Y -135.759,Z 225.711,A 30.186,B 90.000,C 0.000} C_DIS
LIN {X -248.946,Y -144.810,Z 225.711,A 30.186,B 90.000,C 0.000} C_DIS
LIN {X -250.675,Y -145.815,Z 225.711,A 30.186,B 90.000,C 0.000} C_DIS
WAIT SEC 1.75
RET=EKI_SetBool("oxy","torchState",TRUE)
RET = EKI_Send("oxy","torchState")
LIN {X -249.409,Y -147.969,Z 225.794,A 30.680,B 90.000,C 0.000} C_DIS
LIN {X -248.125,Y -150.112,Z 225.892,A 31.173,B 90.000,C 0.000} C_DIS
LIN {X -246.822,Y -152.242,Z 226.002,A 31.667,B 90.000,C 0.000} C_DIS
LIN {X -245.501,Y -154.361,Z 226.124,A 32.160,B 90.000,C 0.000} C_DIS
LIN {X -244.162,Y -156.468,Z 226.255,A 32.653,B 90.000,C 0.000} C_DIS
LIN {X -242.807,Y -158.564,Z 226.394,A 33.146,B 90.000,C 0.000} C_DIS
LIN {X -241.435,Y -160.648,Z 226.540,A 33.639,B 90.000,C 0.000} C_DIS
LIN {X -240.039,Y -162.716,Z 226.692,A 34.132,B 90.000,C 0.000} C_DIS
LIN {X -238.636,Y -164.779,Z 226.847,A 34.625,B 90.000,C 0.000} C_DIS
LIN {X -237.209,Y -166.825,Z 227.006,A 35.118,B 90.000,C 0.000} C_DIS
LIN {X -235.764,Y -168.859,Z 227.165,A 35.611,B 90.000,C 0.000} C_DIS
LIN {X -234.299,Y -170.878,Z 227.323,A 36.104,B 90.000,C 0.000} C_DIS
LIN {X -232.824,Y -172.890,Z 227.481,A 36.597,B 90.000,C 0.000} C_DIS
LIN {X -231.329,Y -174.887,Z 227.635,A 37.090,B 90.000,C 0.000} C_DIS
LIN {X -229.816,Y -176.872,Z 227.785,A 37.583,B 90.000,C 0.000} C_DIS
LIN {X -228.287,Y -178.844,Z 227.928,A 38.076,B 90.000,C 0.000} C_DIS
LIN {X -226.738,Y -180.801,Z 228.064,A 38.569,B 90.000,C 0.000} C_DIS
LIN {X -225.171,Y -182.744,Z 228.189,A 39.062,B 90.000,C 0.000} C_DIS
LIN {X -223.590,Y -184.677,Z 228.306,A 39.555,B 90.000,C 0.000} C_DIS
LIN {X -221.992,Y -186.597,Z 228.411,A 40.049,B 90.000,C 0.000} C_DIS
LIN {X -220.378,Y -188.503,Z 228.502,A 40.542,B 90.000,C 0.000} C_DIS
LIN {X -218.746,Y -190.395,Z 228.579,A 41.036,B 90.000,C 0.000} C_DIS
LIN {X -217.097,Y -192.273,Z 228.638,A 41.530,B 90.000,C 0.000} C_DIS
LIN {X -215.431,Y -194.136,Z 228.680,A 42.024,B 90.000,C 0.000} C_DIS
LIN {X -213.750,Y -195.986,Z 228.702,A 42.518,B 90.000,C 0.000} C_DIS
LIN {X -212.052,Y -197.820,Z 228.703,A 43.011,B 90.000,C 0.000} C_DIS
LIN {X -210.419,Y -199.559,Z 228.686,A 43.483,B 90.000,C 0.000} C_DIS
LIN {X -208.968,Y -198.182,Z 228.686,A 43.483,B 90.000,C 0.000} C_DIS
WAIT SEC 0.1
RET=EKI_SetBool("oxy","torchState",FALSE)
RET = EKI_Send("oxy","torchState")
LIN {X -195.908,Y -185.796,Z 228.686,A 43.483,B 90.000,C 0.000} C_DIS
LIN {X -180.278,Y -200.997,Z 228.355,A 48.110,B 90.000,C 0.000} C_DIS
LIN {X -192.297,Y -214.396,Z 228.355,A 48.110,B 90.000,C 0.000} C_DIS
LIN {X -193.632,Y -215.885,Z 228.355,A 48.110,B 90.000,C 0.000} C_DIS
WAIT SEC 1.75
RET=EKI_SetBool("oxy","torchState",TRUE)
RET = EKI_Send("oxy","torchState")
LIN {X -191.765,Y -217.545,Z 228.445,A 48.604,B 90.000,C 0.000} C_DIS
LIN {X -189.885,Y -219.187,Z 228.578,A 49.097,B 90.000,C 0.000} C_DIS
LIN {X -187.994,Y -220.812,Z 228.753,A 49.590,B 90.000,C 0.000} C_DIS
LIN {X -186.091,Y -222.418,Z 228.976,A 50.082,B 90.000,C 0.000} C_DIS
LIN {X -184.178,Y -224.005,Z 229.240,A 50.573,B 90.000,C 0.000} C_DIS
LIN {X -182.255,Y -225.572,Z 229.548,A 51.063,B 90.000,C 0.000} C_DIS
LIN {X -180.324,Y -227.119,Z 229.902,A 51.552,B 90.000,C 0.000} C_DIS
LIN {X -178.384,Y -228.645,Z 230.298,A 52.039,B 90.000,C 0.000} C_DIS
LIN {X -176.438,Y -230.151,Z 230.736,A 52.526,B 90.000,C 0.000} C_DIS
